// TIA Portal project "planta1_def_V15_V15.1" (V15.1)

(* hardware
DEVICE "S71500/ET200MP station_1"  S7-1500 station
   slot 0: "Perfil soporte_0"  Rack  6ES7 590-1***0-0AA0
   slot 1: "PLC_1"  CPU 1516-3 PN/DP  6ES7 516-3AN00-0AB0  V1.7
   slot 2: "DI 32x24VDC HF_1"  DI 32x24VDC HF  6ES7 521-1BL00-0AB0  V2.0
   slot 3: "DQ 32x24VDC/0.5A ST_1"  DQ 32x24VDC/0.5A ST  6ES7 522-1BL00-0AB0  V2.0
   slot 4: "AI 8xU/I/RTD/TC ST_1"  AI 8xU/I/RTD/TC ST  6ES7 531-7KF00-0AB0  V2.0
   slot 5: "AQ 4xU/I ST_1"  AQ 4xU/I ST  6ES7 532-5HD00-0AB0  V2.0
DEVICE "HMI_1"  TP1500 Comfort
   slot 0: "HMI"  HMI  6AV2 124-0QC02-0AX0  13.0.1.0
   slot 1: "HMI_RT_1"  TP1500 Comfort  6AV2 124-0QC02-0AX0  13.0.1.0
   slot 5: "HMI_1.IE_CP_1"  Interfaz PROFINET
      slot 1: "Interfaz PROFINET_1"  Interfaz PROFINET
         slot 1: "Port_1"  Port
         slot 2: "Port_2"  Port
   slot 6: "HMI_1.IE_CP_2"  Interfaz PROFINET
      slot 1: "Interfaz PROFINET_GBit"  Interfaz PROFINET
         slot 1: "Port_1"  Port
   slot 7: "HMI_1.MPI/DP_CP_1"  Interfaz MPI/DP
*)

// ===== PLC "PLC_1"  CPU 1516-3 PN/DP =====

VAR_GLOBAL   // PLC tag table "Tabla de variables estándar"
   "Switch de Nivel Bajo Tanque 1 (NO)" AT %I1.2 : Bool;   // OK
   "Switch de Nivel Alto Tanque 1 (NC)" AT %I1.3 : Bool;   // OK
   "Referencia Velocidad (VV)" AT %IW104 : Int;   // OK
   "Temperatura Liquido" AT %IW106 : Int;   // OK
   "Presión Liquido" AT %IW108 : Int;   // OK
   "Flujo Actual" AT %IW110 : Int;   // OK
   "Nivel tanque" AT %IW112 : Int;
   "Peso" AT %IW114 : Int;
   "FALLA (VF_DO2)" AT %I2.1 : Bool;   // Sin probar
   "Confirmación Celda BW31" AT %I2.6 : Bool;   // OK (Piloto por revisar)
   "ON/OFF1 (VF_DI1)" AT %Q2.0 : Bool;   // OK
   "Inversión (VF_DI2)" AT %Q2.1 : Bool;
   "Confirmación de Fallo (VF_DI3)" AT %Q2.2 : Bool;
   "Activar Unidad Calefactora" AT %Q1.6 : Bool;
   "RST Total1 (TF01)" AT %Q2.4 : Bool;   // OK
   "Siwarex DI0" AT %Q2.6 : Bool;
   "Siwarex DI1" AT %Q2.7 : Bool;
   "Abrir Valvula Llenado Tanque 1" AT %Q1.0 : Bool;   // OK
   "Abrir Valvula Vaciado Tanque 1" AT %Q1.1 : Bool;   // OK
   "Abrir Valvula Llenado Tanque 2" AT %Q1.2 : Bool;   // OK
   "Abrir Valvula Vaciado Tanque 2" AT %Q1.3 : Bool;   // OK
   "Abrir Valvula Llenado Tanque 3" AT %Q1.4 : Bool;   // OK
   "Abrir Valvula Vaciado Tanque 3" AT %Q1.5 : Bool;
   "Activar Unidad Enfriadora" AT %Q1.7 : Bool;   // OK
   "Panel de Mandos - Display 1" AT %QW100 : Int;
   "Panel de Mandos - Display 2" AT %QW102 : Int;
   "Consigna Velocidad Variador" AT %QW104 : Int;   // OK
   "Consigna apertura Valvula Proporcional" AT %QW106 : Int;   // OK
   "JOG Adelante (VF_DI4)" AT %Q2.3 : Bool;
   "System_Byte" AT %MB1 : Byte;
   "FirstScan" AT %M1.0 : Bool;
   "DiagStatusUpdate" AT %M1.1 : Bool;
   "AlwaysTRUE" AT %M1.2 : Bool;
   "AlwaysFALSE" AT %M1.3 : Bool;
   "Clock_Byte" AT %MB0 : Byte;
   "Clock_10Hz" AT %M0.0 : Bool;
   "Clock_5Hz" AT %M0.1 : Bool;
   "Clock_2.5Hz" AT %M0.2 : Bool;
   "Clock_2Hz" AT %M0.3 : Bool;
   "Clock_1.25Hz" AT %M0.4 : Bool;
   "Clock_1Hz" AT %M0.5 : Bool;
   "Clock_0.625Hz" AT %M0.6 : Bool;
   "Clock_0.5Hz" AT %M0.7 : Bool;
   "bomba" AT %MW6 : Int;
   "valvula" AT %MW8 : Int;
   "v1llen" AT %M2.3 : Bool;
   "v1vac" AT %M2.4 : Bool;
   "v2llen" AT %M2.5 : Bool;
   "v2vac" AT %M2.6 : Bool;
   "onproc" AT %M2.7 : Bool;
   "v3 vac" AT %M5.0 : Bool;
   "d7" AT %M3.0 : Bool;
   "presion" AT %MD10 : Real;
   "flujo" AT %MD14 : Real;
   "dfdf" AT %MD18 : Real;
   "encenderr" AT %M3.1 : Bool;
   "velmotor" AT %MW26 : Word;
   "Tag_19" AT %M3.2 : Bool;
   "onfuzz" AT %M5.1 : Bool;
   "onsint" AT %M5.3 : Bool;
   "onsmith" AT %M5.4 : Bool;
   "refsm" AT %MD20 : Real;
   "reffuzz" AT %MD22 : Real;
   "refsint" AT %MD24 : Real;
   "onsmtant" AT %M5.5 : Bool;
   "onlgr" AT %M5.6 : Bool;
   "reflgr" AT %MD26 : Real;
   "refsmtant" AT %MD28 : Real;
   "calefactora" AT %M6.0 : Bool;
   "Tag_21" AT %M6.1 : Bool;
   "enfriadora" AT %M7.0 : Bool;
   "temperatura" AT %MD16 : Real;
   "on_temp" AT %M5.7 : Bool;
   "REFTEMP" AT %MD30 : Real;
   "v3 llen" AT %M8.0 : Bool;
   "Tag_24" AT %MD50 : Real;
   "kp_sint" AT %MD34 : Real;
   "ki_sint" AT %MD38 : Real;
   "kd_sint" AT %MD42 : Real;
   "kp_lgr" AT %MD46 : Real;
   "ki_lgr" AT %MD54 : Real;
   "kd_lgr" AT %MD58 : Real;
   "kp_smith" AT %MD62 : Real;
   "ki_smith" AT %MD66 : Real;
   "kd_smith" AT %MD70 : Real;
   "kp_smitant" AT %MD74 : Real;
   "ki_smitant" AT %MD78 : Real;
   "kd_smitant" AT %MD82 : Real;
   "CERO_FUZ" AT %MD86 : Real;
   "POS_FUZZ" AT %MD90 : Real;
   "NEG_FUZZ" AT %MD94 : Real;
   "EN_1" AT %MD98 : Real;
   "EN_2" AT %MD102 : Real;
   "EN_3" AT %MD106 : Real;
   "EN_4" AT %MD110 : Real;
   "DEN_1" AT %MD114 : Real;
   "DEN_2" AT %MD118 : Real;
   "DEN_3" AT %MD122 : Real;
   "DEN_4" AT %MD126 : Real;
   "EZ_1" AT %MD130 : Real;
   "EZ_2" AT %MD134 : Real;
   "EZ_3" AT %MD138 : Real;
   "EZ_4" AT %MD142 : Real;
   "DEZ_1" AT %MD146 : Real;
   "DEZ_2" AT %MD150 : Real;
   "DEZ_3" AT %MD154 : Real;
   "DEZ_4" AT %MD158 : Real;
   "EP_1" AT %MD162 : Real;
   "EP_2" AT %MD166 : Real;
   "EP_3" AT %MD170 : Real;
   "EP_4" AT %MD174 : Real;
   "DEP_1" AT %MD178 : Real;
   "DEP_2" AT %MD182 : Real;
   "DEP_3" AT %MD186 : Real;
   "VARIADORFUZZ" AT %MD190 : Real;
   "DEP_4" AT %MD194 : Real;
   "ref_sint_presion" AT %MD198 : Real;
   "kp_sint_pres" AT %MD202 : Real;
   "ki_sint_presion" AT %MD206 : Real;
   "kd_sint_presion" AT %MD210 : Real;
   "on_sint_presion" AT %M2.0 : Bool;
   "on_lgr_flujo" AT %M2.1 : Bool;
   "ref_lgr_flujo" AT %MD214 : Real;
   "kp_lgr_flujo" AT %MD218 : Real;
   "ki_lgr_flujo" AT %MD222 : Real;
   "kd_lgr_flujo" AT %MD226 : Real;
   "onfuzz_presion" AT %M2.2 : Bool;
   "CERO_FUZ_presion" AT %MD230 : Real;
   "POS_FUZZ_presion" AT %MD234 : Real;
   "NEG_FUZZ_presion" AT %MD238 : Real;
   "EN_1_presion" AT %MD242 : Real;
   "EN_2_presion" AT %MD246 : Real;
   "EN_3_presion" AT %MD250 : Real;
   "EN_4_presion" AT %MD254 : Real;
   "DEN_1_presion" AT %MD258 : Real;
   "DEN_2_presion" AT %MD262 : Real;
   "DEN_3_presion" AT %MD266 : Real;
   "DEN_4_presion" AT %MD270 : Real;
   "EZ_1_presion" AT %MD274 : Real;
   "EZ_2_presion" AT %MD278 : Real;
   "EZ_3_presion" AT %MD282 : Real;
   "EZ_4_presion" AT %MD286 : Real;
   "DEZ_1_presion" AT %MD290 : Real;
   "DEZ_2_presion" AT %MD294 : Real;
   "DEZ_3_presion" AT %MD298 : Real;
   "DEZ_4_presion" AT %MD302 : Real;
   "EP_1_presion" AT %MD306 : Real;
   "EP_2_presion" AT %MD310 : Real;
   "EP_3_presion" AT %MD314 : Real;
   "EP_4_presion" AT %MD318 : Real;
   "DEP_1_presion" AT %MD322 : Real;
   "DEP_2_presion" AT %MD326 : Real;
   "DEP_3_presion" AT %MD330 : Real;
   "VARIADORFUZZ_presion" AT %MD334 : Real;
   "DEP_4_presion" AT %MD338 : Real;
   "reffuzz_presion" AT %MD342 : Real;
   "nivel_tanque" AT %MD346 : Real;
   "on_lgr_nivel" AT %M3.3 : Bool;
   "ref_lgr_nivel" AT %MD350 : Real;
   "kp_lgr_nivel" AT %MD354 : Real;
   "ki_lgr_nivel" AT %MD358 : Real;
   "kd_lgr_nivel" AT %MD362 : Real;
   "ALARMA1" AT %M200.0 : Bool;
   "ALARMA2" AT %M200.1 : Bool;
   "ALARMA3" AT %M200.3 : Bool;
   "on_nivel" AT %M3.4 : Bool;
   "ref_onoff_nivel" AT %MD366 : Real;
   "on_peso" AT %M3.5 : Bool;
   "peso tanque" AT %MD370 : Real;
   "ref_onoff_peso" AT %MD374 : Real;
   "Tag_1" AT %I2.3 : Bool;
   "Tag_2" AT %Q2.5 : Bool;
   "enclavar" AT %M3.6 : Bool;
   "Tag_3" AT %MW120 : Word;
   "Tag_4" AT %MD378 : Real;
   "Tag_5" AT %M100.4 : Bool;
   "Tag_6" AT %M100.5 : Bool;
   "Tag_7" AT %M100.6 : Bool;
   "M_Caracterizaicon" AT %M3.7 : Bool;
   "flujo_cal" AT %MD382 : Real;
   "presion_cal" AT %MD386 : Real;
   "temperatura_cal" AT %MD390 : Real;
   "nivel_cal" AT %MD394 : Real;
   "llenadot2" AT %M4.0 : Bool;
   "consigna_variador" AT %MW398 : Int;
   "iniciar_presion" AT %M4.1 : Bool;
   "llenadot1" AT %M4.2 : Bool;
   "ini_flujo" AT %M4.3 : Bool;
   "ini_temp" AT %M4.4 : Bool;
   "INICIAR_PID" AT %M4.5 : Bool;
   "sensor" AT %IW4 : Int;
   "sensor(1)" AT %IW6 : Int;
   "sensor(2)" AT %MW400 : Int;
   "act_calefactora" AT %M4.6 : Bool;
   "referen1" AT %MD402 : Real;
   "INICIAR_PIDP" AT %M4.7 : Bool;
   "Tag_8" AT %M33.0 : Bool;
   "Tag_9" AT %M18.1 : Bool;
   "Tag_10" AT %M18.2 : Bool;
   "Tag_11" AT %MD5 : Real;
   "Tag_12" AT %M71.0 : Bool;
   "Tag_13" AT %M12.0 : Bool;
   "Tag_14" AT %T1 : Timer;
   "Start" AT %M406.0 : Bool;
   "Tag_15" AT %M14.0 : Bool;
   "Tag_16" AT %M1.5 : Bool;
   "Tag_17" AT %QW20 : Word;
   "Tag_18" AT %MW20 : Word;
   "Tag_20" AT %T2 : Timer;
   "Tag_22" AT %MD100 : DWord;
   "Tag_23" AT %Q8.0 : Bool;
   "Tag_25" AT %MD101 : DWord;
   "Tag_26" AT %I2.0 : Bool;
   "Tag_27" AT %MD200 : Time;
   "Tag_28" AT %MD201 : Time;
   "Tag_29" AT %MD300 : Time;
   "Tag_30" AT %MD301 : Time;
   "activacion" AT %M406.1 : Bool;
   "u1" AT %MD408 : Real;
   "u2" AT %MD412 : Real;
   "e1" AT %MD416 : Real;
   "e2" AT %MD420 : Real;
   "rrr" AT %MD424 : Real;
   "activacion_smith_flujo" AT %M406.2 : Bool;
   "u3" AT %MD428 : Real;
   "u4" AT %MD432 : Real;
   "e3" AT %MD436 : Real;
   "e4" AT %MD440 : Real;
   "u1_1" AT %MD444 : Real;
   "u2_1" AT %MD448 : Real;
   "e1_1" AT %MD452 : Real;
   "e2_1" AT %MD456 : Real;
   "activacion_presion_si_es" AT %M406.3 : Bool;
   "referencia_fujo" AT %MD460 : Real;
   "activacion_filtro" AT %M406.4 : Bool;
   "presion_filtrada" AT %MD464 : Real;
   "e1f" AT %MD468 : Real;
   "e2f" AT %MD472 : Real;
   "u1f" AT %MD476 : Real;
   "u2f" AT %MD480 : Real;
   "activacion_flujo_definitivo" AT %M406.5 : Bool;
   "ref_presion" AT %MD484 : Real;
   "u11" AT %MD488 : Real;
   "u22" AT %MD492 : Real;
   "u33" AT %MD496 : Real;
   "u44" AT %MD500 : Real;
   "e11" AT %MD504 : Real;
   "e22" AT %MD508 : Real;
   "e33" AT %MD512 : Real;
   "e44" AT %MD516 : Real;
END_VAR

DATA_BLOCK "lgr_DB_1"   // DB1
{ S7_Optimized_Access := 'TRUE' }
VERSION : 0.1
// stored: InstanceOfName lgr
"lgr"
BEGIN
END_DATA_BLOCK

DATA_BLOCK "sintonizacion_DB_1"   // DB2
{ S7_Optimized_Access := 'TRUE' }
VERSION : 0.1
// stored: InstanceOfName sintonizacion
"sintonizacion"
BEGIN
END_DATA_BLOCK

DATA_BLOCK "smith_DB_2"   // DB3
{ S7_Optimized_Access := 'TRUE' }
VERSION : 0.1
// stored: InstanceOfName smith
"smith"
BEGIN
END_DATA_BLOCK

DATA_BLOCK "smithanticipativo_DB_1"   // DB4
{ S7_Optimized_Access := 'TRUE' }
VERSION : 0.1
// stored: InstanceOfName smithanticipativo
"smithanticipativo"
BEGIN
END_DATA_BLOCK

DATA_BLOCK "principal_DB"   // DB5
{ S7_Optimized_Access := 'TRUE' }
VERSION : 0.1
// stored: InstanceOfName principal
"principal"
BEGIN
END_DATA_BLOCK

DATA_BLOCK "lgr_DB_2"   // DB6
{ S7_Optimized_Access := 'TRUE' }
VERSION : 0.1
// stored: InstanceOfName lgr
"lgr"
BEGIN
END_DATA_BLOCK

DATA_BLOCK "ALARMA"   // DB7
{ S7_Optimized_Access := 'TRUE' }
VERSION : 0.1
   VAR
      ALARMA1 : Int;
      ALARMA2 : Int;
      ALARMA3 : Int;
      ALARMA4 : Int;
      ALARMA5 : Int;
      ALARMA6 : Int;
      ALARMA7 : Int;
      ALARMA8 : Int;
      ALARMA9 : Int;
      ALARMA10 : Int;
      ALARMA11 : Int;
      ALARMA12 : Int;
      ALARMA13 : Int;
      ALARMA14 : Int;
      ALARMA15 : Int;
      ALARMA16 : Int;
      ALARMA17 : Int;
      ALARMA18 : Int;
      ALARMA19 : Int;
      ALARMA20 : Int;
      ALARMA21 : Int;
      ALARMA22 : Int;
   END_VAR
BEGIN
END_DATA_BLOCK

DATA_BLOCK "DATOS_ENTRADAS_ANALOGAS"   // DB8
{ S7_Optimized_Access := 'TRUE' }
VERSION : 0.1
   VAR RETAIN
      "TRANSMISOR DE CAUDAL" : Struct   // Corriente 4 a 20 mA, 0 a 2000 l/h
         "LIMITE SUPERIOR" : Real := 2000.0;
         "LIMITE INFERIOR" : Real;
         AJUSTE : Real;
         "PUNTO INFERIOR" : Real;
         SOBRELIMITE : Bool;
         "ROTURA HILO" : Bool;
         "SEÑAL INGENIERIA" : Real;
      END_STRUCT;
      "TRANSMISOR DE PRESION" : Struct   // Corriente 4 a 20 mA, 0 a 36,25 psi
         "LIMITE SUPERIOR" : Real := 36.2594;   // 2,5 Bar = 36,2594 psi
         "LIMITE INFERIOR" : Real;
         AJUSTE : Real;
         "PUNTO INFERIOR" : Real;
         SOBRELIMITE : Bool;
         "ROTURA HILO" : Bool;
         "SEÑAL INGENIERIA" : Real;
      END_STRUCT;
      "TRANSMISOR DE TEMPERATURA" : Struct
         "LIMITE SUPERIOR" : Real := 100.0;
         "LIMITE INFERIOR" : Real;
         AJUSTE : Real;
         "PUNTO INFERIOR" : Real;
         SOBRELIMITE : Bool;
         "ROTURA HILO" : Bool;
         "SEÑAL INGENIERIA" : Real;
      END_STRUCT;
      "TRANSMISOR DE NIVEL" : Struct
         "LIMITE SUPERIOR" : Real := 100.0;
         "LIMITE INFERIOR" : Real;
         AJUSTE : Real;
         "PUNTO INFERIOR" : Real;
         SOBRELIMITE : Bool;
         "ROTURA HILO" : Bool;
         "SEÑAL INGENIERIA" : Real;
      END_STRUCT;
      "POTENCIOMETRO 1" : Struct   // Corriente 0 a 20 mA
         "LIMITE SUPERIOR" : Real := 20.0;
         "LIMITE INFERIOR" : Real;
         AJUSTE : Real;
         "PUNTO INFERIOR" : Real;
         SOBRELIMITE : Bool;
         "ROTURA HILO" : Bool;
         "SEÑAL INGENIERIA" : Real;
      END_STRUCT;
      "POTENCIOMETRO 2" : Struct   // Voltaje 0 a 10 V
         "LIMITE SUPERIOR" : Real := 10.0;
         "LIMITE INFERIOR" : Real;
         AJUSTE : Real;
         "PUNTO INFERIOR" : Real;
         SOBRELIMITE : Bool;
         "ROTURA HILO" : Bool;
         "SEÑAL INGENIERIA" : Real;
      END_STRUCT;
      VELOCIDAD_VARIADOR : Struct   // Corriente 4 a 20 mA, 0 a 100%
         "LIMITE SUPERIOR" : Real := 100.0;
         "LIMITE INFERIOR" : Real;
         AJUSTE : Real;
         "PUNTO INFERIOR" : Real;
         SOBRELIMITE : Bool;
         "ROTURA HILO" : Bool;
         "SEÑAL INGENIERIA" : Real;
      END_STRUCT;
   END_VAR
   VAR
      PESO : Struct   // Corriente 0 a 20 mA, 0 a 1,4 kg
         "LIMITE SUPERIOR" : Real := 1400.0;
         "LIMITE INFERIOR" : Real;
         AJUSTE : Real;
         "PUNTO INFERIOR" : Real;
         SOBRELIMITE : Bool;
         "ROTURA HILO" : Bool;
         "SEÑAL INGENIERIA" : Real;
      END_STRUCT;
   END_VAR
BEGIN
END_DATA_BLOCK

DATA_BLOCK "OnOff_nivel_DB"   // DB9
{ S7_Optimized_Access := 'TRUE' }
VERSION : 0.1
// stored: InstanceOfName OnOff_nivel
"OnOff_nivel"
BEGIN
END_DATA_BLOCK

DATA_BLOCK "DATOS_SALIDAS_ANALOGAS"   // DB10
{ S7_Optimized_Access := 'TRUE' }
VERSION : 0.1
   VAR RETAIN
      DISPLAY_1 : Struct
         "LIMITE INFERIOR" : Real := 4.0;
         "LIMITE SUPERIOR" : Real := 20.0;
         SEÑAL_INGENIERIA : Real;
         "REBASE POR EXCESO" : Bool;
      END_STRUCT;
      DISPLAY_2 : Struct
         "LIMITE INFERIOR" : Real;
         "LIMITE SUPERIOR" : Real := 10.0;
         SEÑAL_INGENIERIA : Real;
         "REBASE POR EXCESO" : Bool;
      END_STRUCT;
      "VALVULA PROPORCIONAL" : Struct
         "LIMITE INFERIOR" : Real;
         "LIMITE SUPERIOR" : Real := 100.0;
         SEÑAL_INGENIERIA : Real;
         "REBASE POR EXCESO" : Bool;
      END_STRUCT;
      VARIADOR : Struct
         "LIMITE INFERIOR" : Real;
         "LIMITE SUPERIOR" : Real := 100.0;
         SEÑAL_INGENIERIA : Real;
         "REBASE POR EXCESO" : Bool;
      END_STRUCT;
   END_VAR
BEGIN
END_DATA_BLOCK

DATA_BLOCK "pid NIVEL_DB"   // DB11
{ S7_Optimized_Access := 'TRUE' }
VERSION : 0.1
// stored: InstanceOfName pid NIVEL
"pid NIVEL"
BEGIN
END_DATA_BLOCK

DATA_BLOCK "OnOff_peso_DB"   // DB12
{ S7_Optimized_Access := 'TRUE' }
VERSION : 0.1
// stored: InstanceOfName OnOff_peso
"OnOff_peso"
BEGIN
END_DATA_BLOCK

DATA_BLOCK "VELOCIDAD_VARIADOR_FB_DB"   // DB13
{ S7_Optimized_Access := 'TRUE' }
VERSION : 0.1
// stored: InstanceOfName ENTRADAS_ANALOGAS_FB
"ENTRADAS_ANALOGAS_FB"
BEGIN
END_DATA_BLOCK

DATA_BLOCK "TEMPERATURA_FB_DB"   // DB14
{ S7_Optimized_Access := 'TRUE' }
VERSION : 0.1
// stored: InstanceOfName ENTRADAS_ANALOGAS_FB
"ENTRADAS_ANALOGAS_FB"
BEGIN
END_DATA_BLOCK

DATA_BLOCK "PRESION_LIQUIDO_FB_DB"   // DB15
{ S7_Optimized_Access := 'TRUE' }
VERSION : 0.1
// stored: InstanceOfName ENTRADAS_ANALOGAS_FB
"ENTRADAS_ANALOGAS_FB"
BEGIN
END_DATA_BLOCK

DATA_BLOCK "FLUJO_FB_DB"   // DB16
{ S7_Optimized_Access := 'TRUE' }
VERSION : 0.1
// stored: InstanceOfName ENTRADAS_ANALOGAS_FB
"ENTRADAS_ANALOGAS_FB"
BEGIN
END_DATA_BLOCK

DATA_BLOCK "NIVEL_FB_DB"   // DB17
{ S7_Optimized_Access := 'TRUE' }
VERSION : 0.1
// stored: InstanceOfName ENTRADAS_ANALOGAS_FB
"ENTRADAS_ANALOGAS_FB"
BEGIN
END_DATA_BLOCK

DATA_BLOCK "Caracterizacion_DB_1"   // DB18
{ S7_Optimized_Access := 'TRUE' }
VERSION : 0.1
// stored: InstanceOfName Caracterizacion
"Caracterizacion"
BEGIN
END_DATA_BLOCK

DATA_BLOCK "lgr_DB_3"   // DB19
{ S7_Optimized_Access := 'TRUE' }
VERSION : 0.1
// stored: InstanceOfName lgr
"lgr"
BEGIN
END_DATA_BLOCK

DATA_BLOCK "VELOCIDAD_VARIADOR_QW_FB_DB"   // DB20
{ S7_Optimized_Access := 'TRUE' }
VERSION : 0.1
// stored: InstanceOfName SALIDAS_ANALOGAS_FB
"SALIDAS_ANALOGAS_FB"
BEGIN
END_DATA_BLOCK

DATA_BLOCK "VALVULA_PROPORCIONAL_FB_DB"   // DB21
{ S7_Optimized_Access := 'TRUE' }
VERSION : 0.1
// stored: InstanceOfName SALIDAS_ANALOGAS_FB
"SALIDAS_ANALOGAS_FB"
BEGIN
END_DATA_BLOCK

DATA_BLOCK "Calibracion Flujo_DB_1"   // DB22
{ S7_Optimized_Access := 'TRUE' }
VERSION : 0.1
// stored: InstanceOfName Calibracion Flujo
"Calibracion Flujo"
BEGIN
END_DATA_BLOCK

DATA_BLOCK "lgr_DB_4"   // DB23
{ S7_Optimized_Access := 'TRUE' }
VERSION : 0.1
// stored: InstanceOfName lgr
"lgr"
BEGIN
END_DATA_BLOCK

DATA_BLOCK "Bloque_2_DB"   // DB24
{ S7_Optimized_Access := 'TRUE' }
VERSION : 0.1
// stored: InstanceOfName Bloque_2
"Bloque_2"
BEGIN
END_DATA_BLOCK

DATA_BLOCK "Bloque_2_DB_1"   // DB25
{ S7_Optimized_Access := 'TRUE' }
VERSION : 0.1
// stored: InstanceOfName Bloque_2
"Bloque_2"
BEGIN
END_DATA_BLOCK

DATA_BLOCK "Bloque_2_DB_2"   // DB26
{ S7_Optimized_Access := 'TRUE' }
VERSION : 0.1
// stored: InstanceOfName Bloque_2
"Bloque_2"
BEGIN
END_DATA_BLOCK

DATA_BLOCK "Bloque_2_DB_4"   // DB27
{ S7_Optimized_Access := 'TRUE' }
VERSION : 0.1
// stored: InstanceOfName Bloque_2
"Bloque_2"
BEGIN
END_DATA_BLOCK

DATA_BLOCK "Bloque_2_DB_3"   // DB28
{ S7_Optimized_Access := 'TRUE' }
VERSION : 0.1
// stored: InstanceOfName Bloque_2
"Bloque_2"
BEGIN
END_DATA_BLOCK

DATA_BLOCK "FlujoSergioCortes_DB"   // DB29
{ S7_Optimized_Access := 'TRUE' }
VERSION : 0.1
// stored: InstanceOfName PID_FLUJO
"PID_FLUJO"
BEGIN
END_DATA_BLOCK

DATA_BLOCK "FlujoSergioCortes_DB_1"   // DB30
{ S7_Optimized_Access := 'TRUE' }
VERSION : 0.1
// stored: InstanceOfName PID_FLUJO
"PID_FLUJO"
BEGIN
END_DATA_BLOCK

DATA_BLOCK "Bloque_2_DB_5"   // DB31
{ S7_Optimized_Access := 'TRUE' }
VERSION : 0.1
// stored: InstanceOfName Bloque_2
"Bloque_2"
BEGIN
END_DATA_BLOCK

DATA_BLOCK "Bloque_2_DB_6"   // DB33
{ S7_Optimized_Access := 'TRUE' }
VERSION : 0.1
// stored: InstanceOfName Bloque_2
"Bloque_2"
BEGIN
END_DATA_BLOCK

DATA_BLOCK "PESO_FB_DB"   // DB34
{ S7_Optimized_Access := 'TRUE' }
VERSION : 0.1
// stored: InstanceOfName ENTRADAS_ANALOGAS_FB
"ENTRADAS_ANALOGAS_FB"
BEGIN
END_DATA_BLOCK

DATA_BLOCK "FlujoSergioCortes_DB_2"   // DB35
{ S7_Optimized_Access := 'TRUE' }
VERSION : 0.1
// stored: InstanceOfName PID_FLUJO
"PID_FLUJO"
BEGIN
END_DATA_BLOCK

DATA_BLOCK "Bloque_2_DB_7"   // DB36
{ S7_Optimized_Access := 'TRUE' }
VERSION : 0.1
// stored: InstanceOfName Bloque_2
"Bloque_2"
BEGIN
END_DATA_BLOCK

DATA_BLOCK "fuzzyficacion_DB"   // DB37
{ S7_Optimized_Access := 'TRUE' }
VERSION : 0.1
// stored: InstanceOfName fuzzyficacion
"fuzzyficacion"
BEGIN
END_DATA_BLOCK

DATA_BLOCK "FUZZY"   // DB38
{ S7_Optimized_Access := 'TRUE' }
VERSION : 0.1
// stored: InstanceOfName principal
"principal"
BEGIN
END_DATA_BLOCK

DATA_BLOCK "smith_DB"   // DB39
{ S7_Optimized_Access := 'TRUE' }
VERSION : 0.1
// stored: InstanceOfName smith
"smith"
BEGIN
END_DATA_BLOCK

DATA_BLOCK "smith_DB_1"   // DB40
{ S7_Optimized_Access := 'TRUE' }
VERSION : 0.1
// stored: InstanceOfName smith
"smith"
BEGIN
END_DATA_BLOCK

DATA_BLOCK "smithanticipativo_DB"   // DB41
{ S7_Optimized_Access := 'TRUE' }
VERSION : 0.1
// stored: InstanceOfName smithanticipativo
"smithanticipativo"
BEGIN
END_DATA_BLOCK

DATA_BLOCK "lgr_DB"   // DB42
{ S7_Optimized_Access := 'TRUE' }
VERSION : 0.1
// stored: InstanceOfName lgr
"lgr"
BEGIN
END_DATA_BLOCK

DATA_BLOCK "controltemperatura_DB"   // DB43
{ S7_Optimized_Access := 'TRUE' }
VERSION : 0.1
// stored: InstanceOfName controltemperatura
"controltemperatura"
BEGIN
END_DATA_BLOCK

DATA_BLOCK "FlujoSergioCortes_DB_3"   // DB44
{ S7_Optimized_Access := 'TRUE' }
VERSION : 0.1
// stored: InstanceOfName PID_FLUJO
"PID_FLUJO"
BEGIN
END_DATA_BLOCK

DATA_BLOCK "Calibracion Presion_DB_1"   // DB45
{ S7_Optimized_Access := 'TRUE' }
VERSION : 0.1
// stored: InstanceOfName Calibracion Presion
"Calibracion Presion"
BEGIN
END_DATA_BLOCK

DATA_BLOCK "Calibracion temperatura_DB_1"   // DB46
{ S7_Optimized_Access := 'TRUE' }
VERSION : 0.1
// stored: InstanceOfName Calibracion temperatura
"Calibracion temperatura"
BEGIN
END_DATA_BLOCK

DATA_BLOCK "Calibracion_Nivel_DB_1"   // DB47
{ S7_Optimized_Access := 'TRUE' }
VERSION : 0.1
// stored: InstanceOfName Calibracion_Nivel
"Calibracion_Nivel"
BEGIN
END_DATA_BLOCK

DATA_BLOCK "Caracterizacion_DB"   // DB48
{ S7_Optimized_Access := 'TRUE' }
VERSION : 0.1
// stored: InstanceOfName Caracterizacion
"Caracterizacion"
BEGIN
END_DATA_BLOCK

DATA_BLOCK "Calibracion_Nivel_DB"   // DB49
{ S7_Optimized_Access := 'TRUE' }
VERSION : 0.1
// stored: InstanceOfName Calibracion_Nivel
"Calibracion_Nivel"
BEGIN
END_DATA_BLOCK

DATA_BLOCK "Calibracion Presion_DB"   // DB50
{ S7_Optimized_Access := 'TRUE' }
VERSION : 0.1
// stored: InstanceOfName Calibracion Presion
"Calibracion Presion"
BEGIN
END_DATA_BLOCK

DATA_BLOCK "Calibracion temperatura_DB"   // DB51
{ S7_Optimized_Access := 'TRUE' }
VERSION : 0.1
// stored: InstanceOfName Calibracion temperatura
"Calibracion temperatura"
BEGIN
END_DATA_BLOCK

DATA_BLOCK "Calibracion Flujo_DB"   // DB52
{ S7_Optimized_Access := 'TRUE' }
VERSION : 0.1
// stored: InstanceOfName Calibracion Flujo
"Calibracion Flujo"
BEGIN
END_DATA_BLOCK

DATA_BLOCK "PID_FLUJO_DB"   // DB53
{ S7_Optimized_Access := 'TRUE' }
VERSION : 0.1
// stored: InstanceOfName PID_FLUJO
"PID_FLUJO"
BEGIN
END_DATA_BLOCK

DATA_BLOCK "PID_FLUJO_DB_1"   // DB54
{ S7_Optimized_Access := 'TRUE' }
VERSION : 0.1
// stored: InstanceOfName PID_FLUJO
"PID_FLUJO"
BEGIN
END_DATA_BLOCK

DATA_BLOCK "PID_FLUJO_DB_2"   // DB55
{ S7_Optimized_Access := 'TRUE' }
VERSION : 0.1
// stored: InstanceOfName PID_FLUJO
"PID_FLUJO"
BEGIN
END_DATA_BLOCK

DATA_BLOCK "PID_PRESION_DB"   // DB56
{ S7_Optimized_Access := 'TRUE' }
VERSION : 0.1
// stored: InstanceOfName PID_PRESION
"PID_PRESION"
BEGIN
END_DATA_BLOCK

DATA_BLOCK "smith completo_DB"   // DB57
{ S7_Optimized_Access := 'TRUE' }
VERSION : 0.1
// stored: InstanceOfName smith completo
"smith completo"
BEGIN
END_DATA_BLOCK

DATA_BLOCK "Smith_please_DB"   // DB58
{ S7_Optimized_Access := 'TRUE' }
VERSION : 0.1
// stored: InstanceOfName Smith_please
"Smith_please"
BEGIN
END_DATA_BLOCK

DATA_BLOCK "Smith_please_DB_1"   // DB59
{ S7_Optimized_Access := 'TRUE' }
VERSION : 0.1
// stored: InstanceOfName Smith_please
"Smith_please"
BEGIN
END_DATA_BLOCK

DATA_BLOCK "CAUDAL"   // DB61
{ S7_Optimized_Access := 'TRUE' }
VERSION : 0.1
   VAR
      NIVELT : Array[0..20] of Real;
      NIVELT2 : Array[0..20] of Real;
      FLUJO : Array[0..20] of Real;
   END_VAR
BEGIN
END_DATA_BLOCK

DATA_BLOCK "CALCULO_FLUJO_DB"   // DB65
{ S7_Optimized_Access := 'TRUE' }
VERSION : 0.1
// stored: InstanceOfName CALCULO_FLUJO
"CALCULO_FLUJO"
BEGIN
END_DATA_BLOCK

DATA_BLOCK "DELTA_NIVEL"   // DB66
{ S7_Optimized_Access := 'TRUE' }
VERSION : 0.1
   VAR
      N1 : Real;
      N2 : Real;
      FLUJO : Array[0..50] of Real;
      flujoplc : Array[0..50] of Real;
      DELTA : Real;
   END_VAR
BEGIN
END_DATA_BLOCK

DATA_BLOCK "PresionZd"   // DB69
{ S7_Optimized_Access := 'TRUE' }
VERSION : 0.1
   VAR
      e1 : Real := 0.0;
      e2 : Real := 0.0;
      e3 : Real := 0.0;
      e4 : Real := 0.0;
      e5 : Real := 0.0;
      u1 : Real := 0.0;
      u2 : Real := 0.0;
      u3 : Real := 0.0;
      u4 : Real := 0.0;
      u5 : Real := 0.0;
      ud1 : Real := 0.0;
      ud2 : Real := 0.0;
      ds1 : Real := 0.0;
      ds2 : Real := 0.0;
   END_VAR
BEGIN
END_DATA_BLOCK

DATA_BLOCK "PID_FLUJO_DB_3"   // DB70
{ S7_Optimized_Access := 'TRUE' }
VERSION : 0.1
// stored: InstanceOfName PID_FLUJO
"PID_FLUJO"
BEGIN
END_DATA_BLOCK

DATA_BLOCK "PID_JyH_DB"   // DB71
{ S7_Optimized_Access := 'TRUE' }
VERSION : 0.1
// stored: InstanceOfName PID_JyH
"PID_JyH"
BEGIN
END_DATA_BLOCK

DATA_BLOCK "Smith Flujo_DB"   // DB72
{ S7_Optimized_Access := 'TRUE' }
VERSION : 0.1
// stored: InstanceOfName Smith Flujo
"Smith Flujo"
BEGIN
END_DATA_BLOCK

DATA_BLOCK "Smith Flujo_1_DB"   // DB73
{ S7_Optimized_Access := 'TRUE' }
VERSION : 0.1
// stored: InstanceOfName Smith Presion
"Smith Presion"
BEGIN
END_DATA_BLOCK

DATA_BLOCK "Smith Flujo_DB_1"   // DB74
{ S7_Optimized_Access := 'TRUE' }
VERSION : 0.1
// stored: InstanceOfName Smith Flujo
"Smith Flujo"
BEGIN
END_DATA_BLOCK

DATA_BLOCK "smith_flujo_definitivo_DB"   // DB75
{ S7_Optimized_Access := 'TRUE' }
VERSION : 0.1
// stored: InstanceOfName smith_flujo_definitivo
"smith_flujo_definitivo"
BEGIN
END_DATA_BLOCK

DATA_BLOCK "filto_DB"   // DB76
{ S7_Optimized_Access := 'TRUE' }
VERSION : 0.1
// stored: InstanceOfName filto
"filto"
BEGIN
END_DATA_BLOCK

DATA_BLOCK "smith_presion_definitivo_DB"   // DB77
{ S7_Optimized_Access := 'TRUE' }
VERSION : 0.1
// stored: InstanceOfName smith_presion_definitivo
"smith_presion_definitivo"
BEGIN
END_DATA_BLOCK

// folder: System blocks/Program resources

DATA_BLOCK "IEC_Counter_ml_DB"   // DB32
{ S7_Optimized_Access := 'TRUE' }
AUTHOR : SIMATIC
FAMILY : IEC
NAME : DCNTR
VERSION : 1.2
// stored: InstanceOfName IEC_DCOUNTER
"IEC_DCOUNTER"
BEGIN
END_DATA_BLOCK

DATA_BLOCK "IEC_Timer_0_DB"   // DB60
{ S7_Optimized_Access := 'TRUE' }
AUTHOR : Simatic
FAMILY : IEC
NAME : IEC_TMR
VERSION : 1.0
// stored: InstanceOfName IEC_TIMER
"IEC_TIMER"
BEGIN
END_DATA_BLOCK

DATA_BLOCK "IEC_Timer_0_DB_1"   // DB62
{ S7_Optimized_Access := 'TRUE' }
AUTHOR : Simatic
FAMILY : IEC
NAME : IEC_TMR
VERSION : 1.0
// stored: InstanceOfName IEC_TIMER
"IEC_TIMER"
BEGIN
END_DATA_BLOCK

DATA_BLOCK "IEC_Timer_0_DB_2"   // DB63
{ S7_Optimized_Access := 'TRUE' }
AUTHOR : Simatic
FAMILY : IEC
NAME : IEC_TMR
VERSION : 1.0
// stored: InstanceOfName IEC_TIMER
"IEC_TIMER"
BEGIN
END_DATA_BLOCK

DATA_BLOCK "IEC_Timer_0_DB_3"   // DB64
{ S7_Optimized_Access := 'TRUE' }
AUTHOR : Simatic
FAMILY : IEC
NAME : IEC_TMR
VERSION : 1.0
// stored: InstanceOfName IEC_TIMER
"IEC_TIMER"
BEGIN
END_DATA_BLOCK

DATA_BLOCK "IEC_Timer_0_DB_4"   // DB67
{ S7_Optimized_Access := 'TRUE' }
AUTHOR : Simatic
FAMILY : IEC
NAME : IEC_TMR
VERSION : 1.0
// stored: InstanceOfName IEC_TIMER
"IEC_TIMER"
BEGIN
END_DATA_BLOCK

DATA_BLOCK "IEC_Timer_0_DB_5"   // DB68
{ S7_Optimized_Access := 'TRUE' }
AUTHOR : Simatic
FAMILY : IEC
NAME : IEC_TMR
VERSION : 1.0
// stored: InstanceOfName IEC_TIMER
"IEC_TIMER"
BEGIN
END_DATA_BLOCK

// folder: (top level)

FUNCTION_BLOCK "ENTRADAS_ANALOGAS_FB"   // FB1, LAD
{ S7_Optimized_Access := 'TRUE' }
VERSION : 0.1
   VAR_INPUT
      SEÑAL_PERIFERIA : Int;
      LIMITE_SUPERIOR : Real;
      LIMITE_INFERIOR : Real;
      AJUSTE : Real := 0.0;
      PUNTO_INFERIOR : Real;
   END_VAR
   VAR_OUTPUT
      SEÑAL_INGENIERIA : Real;
      SOBRE_LÍMITE : Bool;
      ROTURA_HILO : Bool;
   END_VAR
   VAR
      SEÑAL_REAL : Real;
      TEMP1 : Real;
      TEMP2 : Real;
      PENDIENTE : Real;
      MX : Real;
      "MX+B" : Real;
      SEÑAL_CORREGIDA : Real;
   END_VAR
BEGIN

REGION Network 1
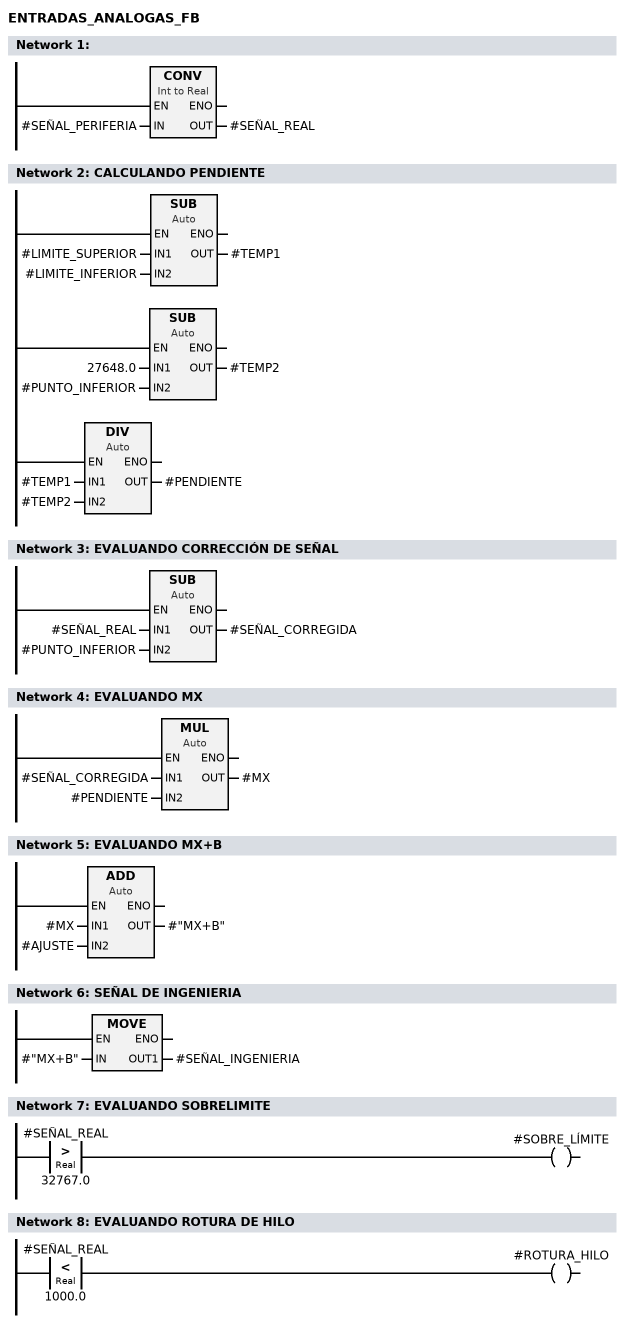
   RUNG wire#powerrail
      { S7_Templates := "[SrcType := Int, DestType := Real]" } Convert(in := #SEÑAL_PERIFERIA, out => #SEÑAL_REAL)
   END_RUNG
   // the same network as SCL:
   #SEÑAL_REAL := INT_TO_REAL(#SEÑAL_PERIFERIA);
END_REGION

REGION Network 2: CALCULANDO PENDIENTE
   RUNG wire#powerrail
      Sub(in1 := #LIMITE_SUPERIOR, in2 := #LIMITE_INFERIOR, out => #TEMP1)
   END_RUNG
   RUNG wire#powerrail
      Sub(in1 := 27648.0, in2 := #PUNTO_INFERIOR, out => #TEMP2)
   END_RUNG
   RUNG wire#powerrail
      Div(in1 := #TEMP1, in2 := #TEMP2, out => #PENDIENTE)
   END_RUNG
   // the same network as SCL:
   #TEMP1 := #LIMITE_SUPERIOR - #LIMITE_INFERIOR;
   #TEMP2 := 27648.0 - #PUNTO_INFERIOR;
   #PENDIENTE := #TEMP1 / #TEMP2;
END_REGION

REGION Network 3: EVALUANDO CORRECCIÓN DE SEÑAL
   RUNG wire#powerrail
      Sub(in1 := #SEÑAL_REAL, in2 := #PUNTO_INFERIOR, out => #SEÑAL_CORREGIDA)
   END_RUNG
   // the same network as SCL:
   #SEÑAL_CORREGIDA := #SEÑAL_REAL - #PUNTO_INFERIOR;
END_REGION

REGION Network 4: EVALUANDO MX
   RUNG wire#powerrail
      Mul(in1 := #SEÑAL_CORREGIDA, in2 := #PENDIENTE, out => #MX)
   END_RUNG
   // the same network as SCL:
   #MX := #SEÑAL_CORREGIDA * #PENDIENTE;
END_REGION

REGION Network 5: EVALUANDO MX+B
   RUNG wire#powerrail
      Add(in1 := #MX, in2 := #AJUSTE, out => #"MX+B")
   END_RUNG
   // the same network as SCL:
   #"MX+B" := #MX + #AJUSTE;
END_REGION

REGION Network 6: SEÑAL DE INGENIERIA
   RUNG wire#powerrail
      Move(in := #"MX+B", out1 => #SEÑAL_INGENIERIA)
   END_RUNG
   // the same network as SCL:
   #SEÑAL_INGENIERIA := #"MX+B";
END_REGION

REGION Network 7: EVALUANDO SOBRELIMITE
   RUNG wire#powerrail
      { S7_Templates := "SrcType := Real" } GT_Contact(in1 := #SEÑAL_REAL, in2 := 32767.0)
      Coil( #SOBRE_LÍMITE )
   END_RUNG
   // the same network as SCL:
   #SOBRE_LÍMITE := #SEÑAL_REAL > 32767.0;
END_REGION

REGION Network 8: EVALUANDO ROTURA DE HILO
   RUNG wire#powerrail
      { S7_Templates := "SrcType := Real" } LT_Contact(in1 := #SEÑAL_REAL, in2 := 1000.0)
      Coil( #ROTURA_HILO )
   END_RUNG
   // the same network as SCL:
   #ROTURA_HILO := #SEÑAL_REAL < 1000.0;
END_REGION
END_FUNCTION_BLOCK

FUNCTION_BLOCK "SALIDAS_ANALOGAS_FB"   // FB2, LAD
{ S7_Optimized_Access := 'TRUE' }
VERSION : 0.1
   VAR_INPUT
      "SEÑAL INGENIERIA" : Real;
      "LIMITE SUPERIOR" : Real;
      "LIMITE INFERIOR" : Real;
      "PUNTO INFERIOR" : Real;
   END_VAR
   VAR_OUTPUT
      "SEÑAL PERIFERIA" : Int;
      "REBASE POR EXCESO" : Bool;
   END_VAR
   VAR_TEMP
      TEMP_1 : Real;
      TEMP_2 : Real;
      TEMP_3 : Real;
      TEMP_4 : Real;
      TEMP_5 : Real;
      K1 : Real;
      K2 : Real;
      SEÑAL_REAL : Real;
   END_VAR
BEGIN

REGION Network 1
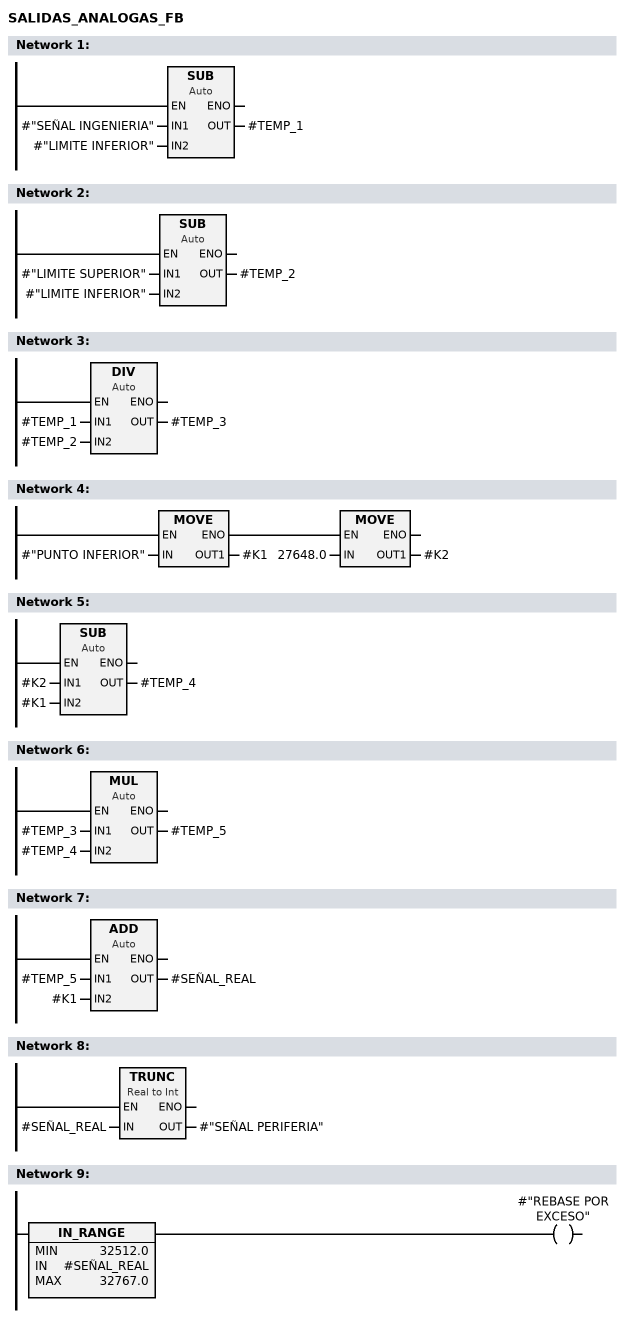
   RUNG wire#powerrail
      Sub(in1 := #"SEÑAL INGENIERIA", in2 := #"LIMITE INFERIOR", out => #TEMP_1)
   END_RUNG
   // the same network as SCL:
   #TEMP_1 := #"SEÑAL INGENIERIA" - #"LIMITE INFERIOR";
END_REGION

REGION Network 2
   RUNG wire#powerrail
      Sub(in1 := #"LIMITE SUPERIOR", in2 := #"LIMITE INFERIOR", out => #TEMP_2)
   END_RUNG
   // the same network as SCL:
   #TEMP_2 := #"LIMITE SUPERIOR" - #"LIMITE INFERIOR";
END_REGION

REGION Network 3
   RUNG wire#powerrail
      Div(in1 := #TEMP_1, in2 := #TEMP_2, out => #TEMP_3)
   END_RUNG
   // the same network as SCL:
   #TEMP_3 := #TEMP_1 / #TEMP_2;
END_REGION

REGION Network 4
   RUNG wire#powerrail
      Move(in := #"PUNTO INFERIOR", out1 => #K1)
      Move(in := 27648.0, out1 => #K2)
   END_RUNG
   // the same network as SCL:
   #K1 := #"PUNTO INFERIOR";
   #K2 := 27648.0;
END_REGION

REGION Network 5
   RUNG wire#powerrail
      Sub(in1 := #K2, in2 := #K1, out => #TEMP_4)
   END_RUNG
   // the same network as SCL:
   #TEMP_4 := #K2 - #K1;
END_REGION

REGION Network 6
   RUNG wire#powerrail
      Mul(in1 := #TEMP_3, in2 := #TEMP_4, out => #TEMP_5)
   END_RUNG
   // the same network as SCL:
   #TEMP_5 := #TEMP_3 * #TEMP_4;
END_REGION

REGION Network 7
   RUNG wire#powerrail
      Add(in1 := #TEMP_5, in2 := #K1, out => #SEÑAL_REAL)
   END_RUNG
   // the same network as SCL:
   #SEÑAL_REAL := #TEMP_5 + #K1;
END_REGION

REGION Network 8
   RUNG wire#powerrail
      { S7_Templates := "[SrcType := Real, DestType := Int]" } Trunc(in := #SEÑAL_REAL, out => #"SEÑAL PERIFERIA")
   END_RUNG
   // the same network as SCL:
   #"SEÑAL PERIFERIA" := TRUNC(#SEÑAL_REAL);
END_REGION

REGION Network 9
   RUNG wire#powerrail
      { S7_Templates := "SrcType := Real" } InRange(min := 32512.0, in := #SEÑAL_REAL, max := 32767.0)
      Coil( #"REBASE POR EXCESO" )
   END_RUNG
   // the same network as SCL:
   #"REBASE POR EXCESO" := (32512.0 <= #SEÑAL_REAL) AND (#SEÑAL_REAL <= 32767.0);
END_REGION
END_FUNCTION_BLOCK

FUNCTION_BLOCK "MAG5100W"   // FB3, LAD
{ S7_Optimized_Access := 'TRUE' }
VERSION : 0.1
   VAR_INPUT
      "Q(ml)" : Bool;
      "OK(Batch)" : Bool;
   END_VAR
   VAR_OUTPUT
      Zero : Bool;
   END_VAR
   VAR
      Reset : Bool;
      FP : Bool;
      Fin_Batch : Bool;
      R_Total_1 : Bool;
      "No(100ml)" : DInt := 10;
      Preset : DInt := 100;
   END_VAR
   VAR_TEMP   // added for the SCL form of the ladder/FBD networks
      _w1 : Bool;
   END_VAR
BEGIN

REGION Network 1
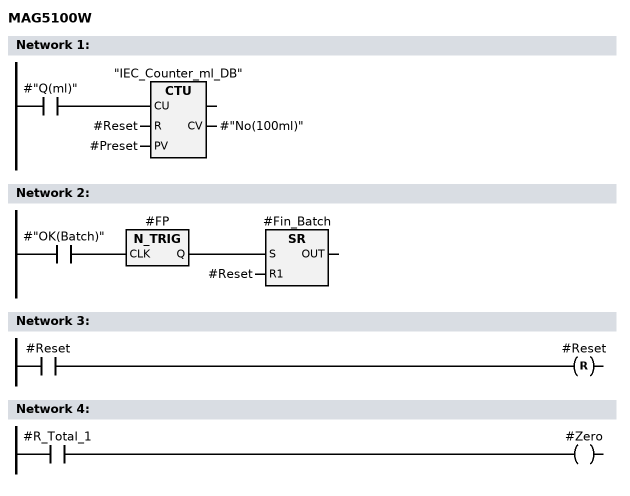
   "IEC_Counter_ml_DB".CTU(CU := #"Q(ml)", R := #Reset, PV := #Preset, CV => #"No(100ml)");
END_REGION

REGION Network 2
   RUNG wire#powerrail
      Contact( #"OK(Batch)" )
      N_Trig( #FP )
      S_SR(operand := #Fin_Batch, r1 := #Reset)
   END_RUNG
   // the same network as SCL:
   #_w1 := NOT #"OK(Batch)" AND #FP;   // falling edge
   #FP := #"OK(Batch)";
   IF #_w1 THEN
       #Fin_Batch := TRUE;   // SR flip-flop
   END_IF;
   IF #Reset THEN #Fin_Batch := FALSE; END_IF;
END_REGION

REGION Network 3
   RUNG wire#powerrail
      Contact( #Reset )
      R_Coil( #Reset )
   END_RUNG
   // the same network as SCL:
   IF #Reset THEN #Reset := FALSE; END_IF;
END_REGION

REGION Network 4
   RUNG wire#powerrail
      Contact( #R_Total_1 )
      Coil( #Zero )
   END_RUNG
   // the same network as SCL:
   #Zero := #R_Total_1;
END_REGION
END_FUNCTION_BLOCK

FUNCTION_BLOCK "sintonizacion"   // FB4, SCL
{ S7_Optimized_Access := 'TRUE' }
VERSION : 0.1
   VAR_INPUT
      ref : Real;
      kp : Real := 30.0;
      ki : Real := 3.0;
      kd : Real := 0.5;
      sensor : Real;
   END_VAR
   VAR_OUTPUT
      señal_u : Real;
      error : Real;
      e0 : Real;
      de : Real;
      e1 : Real;
   END_VAR
BEGIN
   #error := #ref - #sensor;
   #e1 :=  #e1 +#error * 0.01;//periodo de muestreo t
   #de := (#error - #e0) / 0.01;
   //7.2722 49.6172;

   #señal_u := (#kp * #error + #ki * #e1 + #de * #kd);
   IF #señal_u > 27000.0 THEN
       #señal_u := 27000.0;
   END_IF;
   IF #señal_u < 9000.0 THEN
       #señal_u := 9000.0;
   END_IF;
END_FUNCTION_BLOCK

FUNCTION_BLOCK "fuzzyficacion"   // FB5, SCL
{ S7_Optimized_Access := 'TRUE' }
VERSION : 0.1
   VAR_INPUT
      crisp : Real;
      vector1 : Real;
      vector2 : Real;
      vector3 : Real;
      vector4 : Real;
   END_VAR
   VAR_OUTPUT
      S : Real;
   END_VAR
   VAR_TEMP
      "a" : Real;
      "B" : Real;
   END_VAR
BEGIN
   IF (#vector1 < #crisp & #crisp < #vector2) THEN
       #B := -1 * (((1 - 0) / (#vector2 - #vector1)) * #vector1);
       #a := (((1 - 0) / (#vector2 - #vector1)) * #crisp) + #B;
   END_IF;
   IF (#vector2 < #crisp & #crisp < #vector3) THEN
       #a := 1;
   END_IF;
   IF (#vector3 < #crisp & #crisp < #vector4) THEN
       #B := (((1 - 0) / (#vector2 - #vector1)) * #vector4);
       #a := (((0 - 1) / (#vector4 - #vector3)) * #crisp) + #B;
   ELSE
       #a := 0;
   END_IF;
   #S := #a;
END_FUNCTION_BLOCK

FUNCTION_BLOCK "principal"   // FB6, SCL
{ S7_Optimized_Access := 'TRUE' }
VERSION : 0.1
   VAR_INPUT
      sensor : Real;
      ki : Real := 15.0;
      Z : Real := 0.0;
      P : Real := 9730.0;
      N : Real := -9730.0;
      EN1 : Real := -688.0;
      EN2 : Real := -432.0;
      EN3 : Real := -294.8;
      EN4 : Real := -41.3;
      DEN1 : Real := -783.0;
      DEN2 : Real := -607.0;
      DEN3 : Real := -364.1;
      DEN4 : Real := -63.3;
      EZ1 : Real := -103.0;
      EZ2 : Real := -10.0;
      EZ3 : Real := 10.0;
      EZ4 : Real := 104.8;
      DEZ1 : Real := -93.6;
      DEZ2 : Real := -10.4;
      DEZ3 : Real := 10.45;
      DEZ4 : Real := 94.05;
      EP1 : Real := 43.4;
      EP2 : Real := 296.5;
      EP3 : Real := 432.0;
      EP4 : Real := 688.0;
      DEP1 : Real := 11.22;
      DEP2 : Real := 347.0;
      DEP3 : Real := 544.0;
      var : Real := 9000.0;
      DEP4 : Real := 812.0;
      ref : Real;
   END_VAR
   VAR_OUTPUT
      S : Real;
      "e" : Real;
      de : Real;
   END_VAR
   VAR_TEMP
      R1 : Real;
      R2 : Real;
      R3 : Real;
      R4 : Real;
      R5 : Real;
      R6 : Real;
      R7 : Real;
      R8 : Real;
      R9 : Real;
      e0 : Real;
      AA : Real;
      BB : Real;
      eant : Real;
      SS : Real;
      e1 : Real;
      pi : Real;
      CC : Real;
   END_VAR
BEGIN
   #e := #ref - #sensor;
   #de := (#e-#eant);
   #e1 := #e1 + #e;
   #pi := #e1 *#ki;
   #eant := #e;"fuzzyfica"(crisp := #e,
               vector1 := #EN1,
               vector2 := #EN2,
               vector3 := #EN3,
               vector4 := #EN4,
               A_1 => #AA);
   "fuzzyfica" (crisp := #de,
                                     vector1 := #DEN1,
                                     vector2 := #DEN2,
                                     vector3 := #DEN3,
                                     vector4 := #DEN4,
                                     A_1 => #BB);
   #R1:=MIN_REAL(IN1:=#AA,IN2:=#BB);
   "fuzzyfica"(crisp := #e,
                                    vector1 := #EN1,
                                    vector2 := #EN2,
                                    vector3 := #EN3,
                                    vector4 := #EN4,
                                    A_1 => #AA);
   "fuzzyfica"(crisp := #de,
                                    vector1 := #DEZ1,
                                    vector2 := #DEZ2,
                                    vector3 := #DEZ3,
                                    vector4 := #DEZ4,
                                    A_1 => #BB);
   #R2 := MIN_REAL(IN1 := #AA, IN2 := #BB);
   "fuzzyfica"(crisp := #e,
                                    vector1 := #EN1,
                                    vector2 := #EN2,
                                    vector3 := #EN3,
                                    vector4 := #EN4,
                                    A_1 => #AA);
   "fuzzyfica"(crisp := #de,
                                    vector1 := #DEP1,
                                    vector2 := #DEP2,
                                    vector3 := #DEP3,
                                    vector4 := #DEP4,
                                    A_1 => #BB);
   #R3 := MIN_REAL(IN1 := #AA, IN2 := #BB);
   "fuzzyfica"(crisp := #e,
                                    vector1 := #EZ1,
                                    vector2 := #EZ2,
                                    vector3 := #EZ3,
                                    vector4 := #EZ4,
                                    A_1 => #AA);
   "fuzzyfica"(crisp := #de,
                                    vector1 := #DEN1,
                                    vector2 := #DEN2,
                                    vector3 := #DEN3,
                                    vector4 := #DEN4,
                                    A_1 => #BB);
   #R4 := MIN_REAL(IN1 := #AA, IN2 := #BB);
   "fuzzyfica"(crisp := #e,
                                    vector1 := #EZ1,
                                    vector2 := #EZ2,
                                    vector3 := #EZ3,
                                    vector4 := #EZ4,
                                    A_1 => #AA);
   "fuzzyfica"(crisp := #de,
                                    vector1 := #DEZ1,
                                    vector2 := #DEZ2,
                                    vector3 := #DEZ3,
                                    vector4 := #DEZ4,
                                    A_1 => #BB);
   #R5 := MIN_REAL(IN1 := #AA, IN2 := #BB);
   "fuzzyfica"(crisp := #e,
                                    vector1 := #EZ1,
                                    vector2 := #EZ2,
                                    vector3 := #EZ3,
                                    vector4 := #EZ4,
                                    A_1 => #AA);
   "fuzzyfica"(crisp := #de,
                                    vector1 := #DEP1,
                                    vector2 := #DEP2,
                                    vector3 := #DEP3,
                                    vector4 := #DEP4,
                                    A_1 => #BB);
   #R6 := MIN_REAL(IN1 := #AA, IN2 := #BB);
   "fuzzyfica"(crisp := #e,
                                    vector1 := #EP1,
                                    vector2 := #EP2,
                                    vector3 := #EP3,
                                    vector4 := #EP4,
                                    A_1 => #AA);
   "fuzzyfica"(crisp := #de,
                                    vector1 := #DEZ1,
                                    vector2 := #DEZ2,
                                    vector3 := #DEZ3,
                                    vector4 := #DEZ4,
                                    A_1 => #BB);
   #R7 := MIN_REAL(IN1 := #AA, IN2 := #BB);
   "fuzzyfica"(crisp := #e,
                                    vector1 := #EP1,
                                    vector2 := #EP2,
                                    vector3 := #EP3,
                                    vector4 := #EP4,
                                    A_1 => #AA);
   "fuzzyfica"(crisp := #de,
                                    vector1 := #DEP1,
                                    vector2 := #DEP2,
                                    vector3 := #DEP3,
                                    vector4 := #DEP4,
                                    A_1 => #BB);
   #R8 := MIN_REAL(IN1 := #AA, IN2 := #BB);
   "fuzzyfica"(crisp := #e,
                                    vector1 := #EP1,
                                    vector2 := #EP2,
                                    vector3 := #EP3,
                                    vector4 := #EP4,
                                    A_1 => #AA);
   "fuzzyfica"(crisp := #de,
                                    vector1 := #DEN1,
                                    vector2 := #DEN2,
                                    vector3 := #DEN3,
                                    vector4 := #DEN4,
                                    A_1 => #BB);
   #R9 := MIN_REAL(IN1 := #AA, IN2 := #BB);
   #SS := ((#R1 * #N) + (#R2 * #N) + (#R3 * #Z) + (#R4 * #N) + (#R5 * #Z) + (#R6 * #P) + (#R7 * #P) + (#R8 * #P) + (#R9 * #P)) / (#R1 + #R2 + #R3 + #R4 + #R5 + #R6 + #R7 + #R8 + #R9);
   #S := (#var + #SS*1.3)+#pi;
END_FUNCTION_BLOCK

FUNCTION_BLOCK "smith"   // FB7, SCL
{ S7_Optimized_Access := 'TRUE' }
VERSION : 0.1
   VAR_INPUT
      ref : Real;
      refant : Real;
      kp : Real := 154.79;
      ki : Real := 1.083;
      sensorant : Real;
      sensor2ant : Real;
      kd : Real := 0.0;
      variador : Real;
      valprop : Real;
      sensor : Real;
   END_VAR
   VAR_OUTPUT
      u : Real;
      Scy : Real;
      Scy2ant : Real;
      Scyant : Real;
      Scrant : Real;
      Scr : Real;
      cont : Real;
      error : Real;
      e0 : Real;
      de : Real;
      contant : Real;
      "a" : Real;
      bant : Real;
      d : Real;
      c : Real;
      "b" : Real;
      aant : Real;
      ei : Real;
   END_VAR
BEGIN
   #Scr := (1.403*#ref)-(1.397*#refant)+ #Scrant;
   #u := #Scr- #Scy;
   #Scy := (2.932 * #sensor) - (5.857 * #sensorant) + (2.925 * #sensor2ant) + (1.999 * #Scyant) - (0.999 * #Scy2ant);

   #refant := #ref;
   #Scrant := #Scr;
   #sensor2ant := #sensorant;
   #sensorant := #sensor;
   #Scy2ant := #Scyant;
   #Scyant := #Scy;


   IF #u > 27000.0 THEN
       #u := 27000.0;
   END_IF;

   IF #u < 9000.0 THEN
       #u := 9000.0;
   END_IF;
END_FUNCTION_BLOCK

FUNCTION_BLOCK "smithanticipativo"   // FB8, SCL
{ S7_Optimized_Access := 'TRUE' }
VERSION : 0.1
   VAR_INPUT
      ref : Real;
      kp : Real := 154.79;
      ki : Real := 1.083;
      kd : Real := 0.0;
      variador : Real;
      valprop : Real;
      sensor : Real;
   END_VAR
   VAR_OUTPUT
      cont : Real;
      error : Real;
      e0 : Real;
      de : Real;
      contant : Real;
      "a" : Real;
      bant : Real;
      d : Real;
      c : Real;
      "b" : Real;
      aant : Real;
      k : Real;
      j : Real;
      hant : Real;
      h : Real;
      gant : Real;
      g : Real;
      jant : Real;
      kant : Real;
      iant : Real;
      l : Real;
      lant : Real;
      i : Real;
      varant : Real;
      ei : Real;
   END_VAR
BEGIN
   #error := #ref - #j;
   #ei := #ei + #error * 0.01;//periodo de muestreo t
   //#de := (#error - #e0) / 0.01;
   //7.2722 49.6172;
   #cont := (#kp * #error + #ki * #ei);
   #i := (#valprop*-0.002083) + (0.002047*#varant) + (0.9913*#iant);
   #iant := #i;
   #h := (-0.0006298*#i) + (#iant) + (0.0006298*#hant);
   #hant := #h;
   #g := #h + #cont;
   #a := (#g*0.000002235)+(#gant*0.000002235)+(#aant*0.98);
   #b := (#a*-0.9677)+(#aant)+(#bant*0.9677);
   #aant := #a;
   #bant := #b;
   #c:=#sensor-#b;
   #d:=#a+#c;

   (*#l := (#variador*0.000000465) + (#varant*0.000000465) + (0.9914*#lant);
   #lant := #l;
   #k := (-0.9952*#l) + (#lant) + (0.9952*#kant);
   #kant := #k;
   #gant := #g;*)
   #j := #d;
   #contant := #cont;
   #varant := #valprop;
   IF #cont > 27000.0 THEN
       #cont := 27000.0;
   END_IF;
   IF #cont < 9000.0 THEN
       #cont := 9000.0;
   END_IF;
END_FUNCTION_BLOCK

FUNCTION_BLOCK "lgr"   // FB9, SCL
{ S7_Optimized_Access := 'TRUE' }
VERSION : 0.1
   VAR_INPUT
      ref : Real;
      kp : Real := 0.0;
      ki : Real := 0.0;
      kd : Real := 0.0;
      refant : Real;
      sensorant : Real;
      sensor2ant : Real;
      sensor : Real;
   END_VAR
   VAR_OUTPUT
      señal_u : Real;
      Scrant : Real;
      Scyant : Real;
      Scy2ant : Real;
      Scy : Real;
      u : Real;
      Scr : Real;
      Scr2ant : Real;
      error2ant : Real;
      errorant : Real;
      error : Real;
      e0 : Real;
      de : Real;
      e1 : Real;
   END_VAR
BEGIN
   #error := #ref - #sensor;
   //#Scr := (1.4280 * #error) - (1.3623 * #errorant) + #Scrant;

   #Scr := (3071 * #error) - (6138 * #errorant) + (3068* #error2ant) + (1 * #Scr2ant);

   #refant := #ref;
   #Scrant := #Scr;
   #sensor2ant := #sensorant;
   #sensorant := #sensor;
   #Scr2ant := #Scrant;
   #Scrant := #Scy;
   #error2ant := #errorant;
   #errorant := #error;


   IF #Scr > 27000.0 THEN
       #Scr := 27000.0;
   END_IF;

   IF #Scr < 9000.0 THEN
       #Scr := 9000.0;
   END_IF;
END_FUNCTION_BLOCK

FUNCTION_BLOCK "controltemperatura"   // FB10, SCL
{ S7_Optimized_Access := 'TRUE' }
VERSION : 0.1
   VAR_INPUT
      temperatura : Real;
      setpoint : Real;
   END_VAR
   VAR_OUTPUT
      unidadcalentadora : Bool;
      unidadenfriadora : Bool;
   END_VAR
   VAR CONSTANT
      porcentaje : Real;
   END_VAR
BEGIN
   IF #temperatura> #setpoint THEN
       #unidadenfriadora :=1;
       #unidadcalentadora := 0;
   END_IF;
   IF #temperatura < #setpoint THEN
       #unidadenfriadora := 0;
       #unidadcalentadora := 1;
   END_IF;
END_FUNCTION_BLOCK

FUNCTION_BLOCK "OnOff_nivel"   // FB11, SCL
{ S7_Optimized_Access := 'TRUE' }
VERSION : 0.1
   VAR_INPUT
      setpoint : Real;
      sensor : Real;
   END_VAR
   VAR_OUTPUT
      vaciadoT1 : Bool;
      vaciadoT2 : Bool;
      llenadoT1 : Bool;
      llenadoT2 : Bool;
   END_VAR
BEGIN
   IF #sensor > #setpoint THEN
       #vaciadoT1 := 0;
       #vaciadoT2 := 1;
       #llenadoT1 := 1;
       #llenadoT2 := 0;
   END_IF;
   IF #sensor < #setpoint THEN
       #vaciadoT1 := 1;
       #vaciadoT2 := 0;
       #llenadoT1 := 0;
       #llenadoT2 := 1;
   END_IF;
END_FUNCTION_BLOCK

FUNCTION_BLOCK "OnOff_peso"   // FB12, SCL
{ S7_Optimized_Access := 'TRUE' }
VERSION : 0.1
   VAR_INPUT
      setpoint : Real;
      sensor : Real;
   END_VAR
   VAR_OUTPUT
      vaciadoT1 : Bool;
      vaciadoT2 : Bool;
      llenadoT1 : Bool;
      llenadoT2 : Bool;
   END_VAR
BEGIN
   IF #sensor > #setpoint THEN
       #vaciadoT1 := 1;
       #vaciadoT2 := 0;
       #llenadoT1 := 0;
       #llenadoT2 := 1;
   END_IF;
   IF #sensor < #setpoint THEN
       #vaciadoT1 := 0;
       #vaciadoT2 := 1;
       #llenadoT1 := 1;
       #llenadoT2 := 0;
   END_IF;
END_FUNCTION_BLOCK

FUNCTION_BLOCK "pid NIVEL"   // FB13, SCL
{ S7_Optimized_Access := 'TRUE' }
VERSION : 0.1
   VAR_INPUT
      ref : Real;
      kp : Real;
      ki : Real;
      kd : Real;
      sensor : Real;
   END_VAR
   VAR_OUTPUT
      señal_u : Real;
      VACIADOT1 : Bool;
      VACIADOT2 : Bool;
      LLENADOT2 : Bool;
      LLENADOT1 : Bool;
      error : Real;
      e1 : Real;
      de : Real;
      e0 : Real;
   END_VAR
BEGIN
   #error := #ref - #sensor;
   #e1 := #e1 + #error * 0.01;//periodo de muestreo t
   #de := (#error - #e0) / 0.01;
   #señal_u := (#kp * #error + #ki * #e1 + #de * #kd);
   IF #error > 0 THEN
       #VACIADOT1 := 1;
       #VACIADOT2 := 0;
       #LLENADOT1 := 0;
       #LLENADOT2 := 1;
   ELSE
       #VACIADOT1 := 0;
       #VACIADOT2 := 1;
       #LLENADOT1 := 1;
       #LLENADOT2 := 0;
   END_IF;

   IF #señal_u > 27000.0 THEN
       #señal_u := 27000.0;
   END_IF;
   IF #señal_u < 9000.0 THEN
       #señal_u := 9000.0;
   END_IF;
END_FUNCTION_BLOCK

FUNCTION_BLOCK "PID_FLUJO"   // FB14, SCL
{ S7_Optimized_Access := 'TRUE' }
VERSION : 0.1
   VAR_INPUT
      ref : Real;
      sensor : Real;
      rdisturbance : Real;
   END_VAR
   VAR_OUTPUT
      Motor : Real;
      Ojo : Real;
   END_VAR
   VAR_TEMP
      "e" : Real;
      de : Real;
      ie : Real;
      e3 : Real;
      e1 : Real;
      Bomba : Real;
      uc2 : Real;
      u : Real;
      u1 : Real;
      u2 : Real;
      baux : Real;
      e2 : Real;
      ud : Real;
      uc : Real;
      ds : Real;
      uaux : Real;
      eaux : Real;
   END_VAR
   VAR CONSTANT
      ecn : Real := 244.0784;
      ecn1 : Real := 892.0721;
      ecn2 : Real := 1221.698;
      ecn3 : Real := 742.9892;
      ecn4 : Real := 169.2944;
      ucn1 : Real := 3.2507;
      ucn2 : Real := 3.8764;
      ucn3 : Real := 1.9963;
      err2 : Real := 0.0;
      Constant_3 : Real;
      Constant_1 : Real;
      Constant_2 : Real;
      ucn4 : Real := 0.3706;
   END_VAR
BEGIN
   #e := #ref - #sensor;
   //#ds :=27000-  #rdisturbance;
   #Ojo := #e;
   //#u := (#ecn * #e) - (#ecn1 * "PresionZd".e1) + (#ecn2 * "PresionZd".e2) - (#ecn3 * "PresionZd".e3) + (#ecn4 * "PresionZd".e4)
   //+ (#ucn1 * "PresionZd".u1) - (#ucn2 * "PresionZd".u2) + (#ucn3 * "PresionZd".u3) - (#ucn4 * "PresionZd".u4);


   //#ud := 0.2271* #ds -0.4558* "PresionZd".ds1 +0.2281* "PresionZd".ds2
   //+1.909* "PresionZd".ud1 -0.9114*"PresionZd".ud2;
   //
   //#u := (#ecn * #e) - (#ecn1 * "PresionZd".e1) + (#ecn2 * "PresionZd".e2) - (#ecn3 * "PresionZd".e3) + (#ecn4 * "PresionZd".e4)
   //+ (#ucn1 * "PresionZd".u1) - (#ucn2 * "PresionZd".u2) + (#ucn3 * "PresionZd".u3) - (#ucn4 * "PresionZd".u4);
   #u := 148.1*#e-263.9*#e1+117.8*#e2+1.868*#uc-0.8684*#uc2;
   //#u := 76.31 * #e - 143.2 * #e1 + 67.44 * #e2 + 1.874 * #uc - 0.874 * #uc2;

   #uaux := #uc;
   #uc := #u;
   #uc2 := #uaux;

   #baux := #u;//
   #eaux := #e1;
   #e1 := #e;
   #e2 := #eaux;


   IF #baux > 27000.0 THEN
       #Motor := 27000.0;
   ELSIF #baux < 6500.0 THEN
       #Motor := 6500.0;
   ELSE
       #Motor := #baux;
   END_IF;


   //"PresionZd".e4 := "PresionZd".e3;
   //"PresionZd".e3 := "PresionZd".e2;
   //"PresionZd".e2 := "PresionZd".e1;
   //"PresionZd".e1 := #e;

   //"PresionZd".u4 := "PresionZd".u3;
   //"PresionZd".u3 := "PresionZd".u2;
   //"PresionZd".u2 := "PresionZd".u1;
   //"PresionZd".u1 := #u;

   //"PresionZd".ds2 := "PresionZd".ds1;
   //"PresionZd".ds1 := #ds;

   //"PresionZd".ud2 := "PresionZd".ud1;
   //"PresionZd".ud1 := #ud;
END_FUNCTION_BLOCK

FUNCTION_BLOCK "Bloque_2"   // FB15, SCL
{ S7_Optimized_Access := 'TRUE' }
VERSION : 0.1
   VAR_INPUT
      sp : Real;
      y : Real;
      kp : Real;
      ti : Real;
      td : Real;
   END_VAR
   VAR_OUTPUT
      "M" : Real;
   END_VAR
   VAR
      e0 : Real := 0.0;
      e1 : Real;
      de : Real;
      ie : Real;
      ki : Real;
      kd : Real;
   END_VAR
BEGIN
   #e1:=#sp - #y;
   #de := (#e1 - #e0) /  0.01;
   #ie := #ie + (#e1 *  0.01);
   #ki := #kp / #ti;
   #kd:= #kp * #td;
   #M:= #e1*#kp + #ie*#ki +#de*#kd;
   IF #M>32000 THEN
       // Statement section IF
       #M :=32000;
   END_IF;
   IF #M<6500 THEN
       // Statement section IF
       #M := 6500;
   END_IF;

   #e0:=#e1;
END_FUNCTION_BLOCK

FUNCTION_BLOCK "Caracterizacion"   // FB16, LAD
{ S7_Optimized_Access := 'TRUE' }
VERSION : 0.1
   VAR_INPUT
      inicio_llenadot1 : Bool;
      valor_variador : Int;
      valor_valvula : Int;
      inicio_presion : Bool;
      inicio_llenadot2 : Bool;
      inicio_flujo : Bool;
      inicio_temp : Bool;
   END_VAR
   VAR_OUTPUT
      onoff_variador : Bool;
      valv1 : Bool;
      valv2 : Bool;
      valv_pro : Int;
      vaciadot2 : Bool;
      calentador : Bool;
      vaciadot1 : Bool;
   END_VAR
BEGIN

REGION Network 1: medición de nivel tanque 2
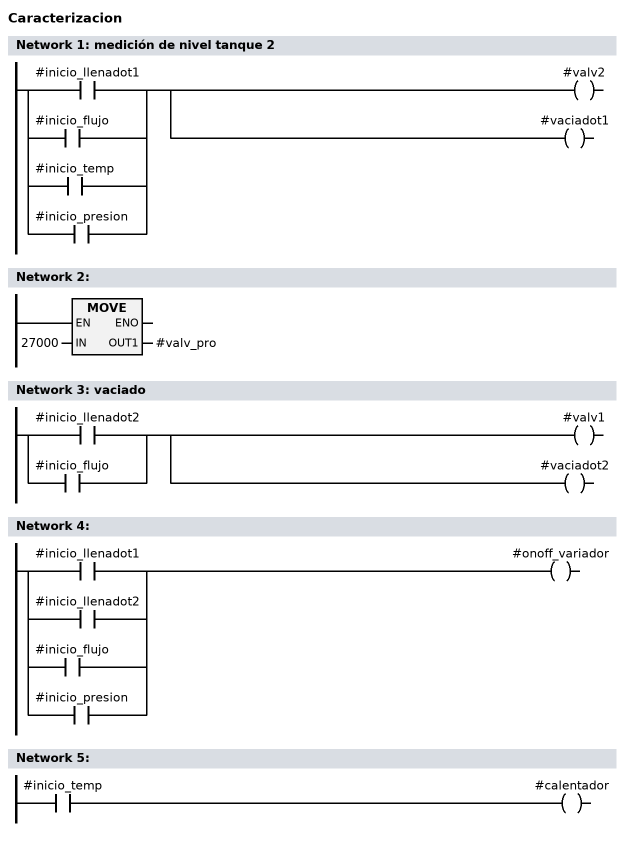
   RUNG wire#powerrail
      Contact( #inicio_llenadot1 )
      wire#w1
      Coil( #valv2 )
   END_RUNG
   RUNG wire#powerrail
      Contact( #inicio_flujo )
   END_RUNG wire#w1
   RUNG wire#powerrail
      Contact( #inicio_temp )
   END_RUNG wire#w1
   RUNG wire#powerrail
      Contact( #inicio_presion )
   END_RUNG wire#w1
   RUNG wire#w1
      Coil( #vaciadot1 )
   END_RUNG
   // the same network as SCL:
   #valv2 := #inicio_llenadot1 OR #inicio_flujo OR #inicio_temp OR #inicio_presion;
   #vaciadot1 := #valv2;
END_REGION

REGION Network 2
   RUNG wire#powerrail
      Move(in := 27000, out1 => #valv_pro)
   END_RUNG
   // the same network as SCL:
   #valv_pro := 27000;
END_REGION

REGION Network 3: vaciado
   RUNG wire#powerrail
      Contact( #inicio_llenadot2 )
      wire#w1
      Coil( #valv1 )
   END_RUNG
   RUNG wire#powerrail
      Contact( #inicio_flujo )
   END_RUNG wire#w1
   RUNG wire#w1
      Coil( #vaciadot2 )
   END_RUNG
   // the same network as SCL:
   #valv1 := #inicio_llenadot2 OR #inicio_flujo;
   #vaciadot2 := #valv1;
END_REGION

REGION Network 4
   RUNG wire#powerrail
      Contact( #inicio_llenadot1 )
      wire#w1
      Coil( #onoff_variador )
   END_RUNG
   RUNG wire#powerrail
      Contact( #inicio_llenadot2 )
   END_RUNG wire#w1
   RUNG wire#powerrail
      Contact( #inicio_flujo )
   END_RUNG wire#w1
   RUNG wire#powerrail
      Contact( #inicio_presion )
   END_RUNG wire#w1
   // the same network as SCL:
   #onoff_variador := #inicio_llenadot1 OR #inicio_llenadot2 OR #inicio_flujo OR #inicio_presion;
END_REGION

REGION Network 5
   RUNG wire#powerrail
      Contact( #inicio_temp )
      Coil( #calentador )
   END_RUNG
   // the same network as SCL:
   #calentador := #inicio_temp;
END_REGION
END_FUNCTION_BLOCK

FUNCTION_BLOCK "Calibracion_Nivel"   // FB17, LAD
{ S7_Optimized_Access := 'TRUE' }
VERSION : 0.1
   VAR_INPUT
      nivTanq : Int;
   END_VAR
   VAR_OUTPUT
      "Ax+B" : Real;
   END_VAR
   VAR
      Ax : Real;
      Static_1 : Real;
   END_VAR
BEGIN

REGION Network 1
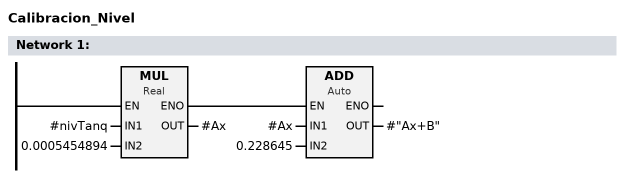
   RUNG wire#powerrail
      { S7_Templates := "SrcType := Real" } Mul(in1 := #nivTanq, in2 := 0.0005454894, out => #Ax)
      Add(in1 := #Ax, in2 := 0.228645, out => #"Ax+B")
   END_RUNG
   // the same network as SCL:
   #Ax := #nivTanq * 0.0005454894;
   #"Ax+B" := #Ax + 0.228645;
END_REGION
END_FUNCTION_BLOCK

FUNCTION_BLOCK "Calibracion Presion"   // FB18, LAD
{ S7_Optimized_Access := 'TRUE' }
VERSION : 0.1
   VAR_INPUT
      presion : Real;
   END_VAR
   VAR_OUTPUT
      "Ax-B" : Real;
   END_VAR
   VAR
      Ax : Real;
   END_VAR
BEGIN

REGION Network 1
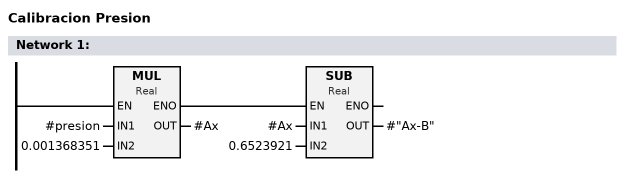
   RUNG wire#powerrail
      { S7_Templates := "SrcType := Real" } Mul(in1 := #presion, in2 := 0.001368351, out => #Ax)
      { S7_Templates := "SrcType := Real" } Sub(in1 := #Ax, in2 := 0.6523921, out => #"Ax-B")
   END_RUNG
   // the same network as SCL:
   #Ax := #presion * 0.001368351;
   #"Ax-B" := #Ax - 0.6523921;
END_REGION
END_FUNCTION_BLOCK

FUNCTION_BLOCK "Calibracion temperatura"   // FB19, LAD
{ S7_Optimized_Access := 'TRUE' }
VERSION : 0.1
   VAR_INPUT
      Temperaturaa : Real;
   END_VAR
   VAR_OUTPUT
      "Ax-B" : Real;
   END_VAR
   VAR
      Ax : Real;
   END_VAR
BEGIN

REGION Network 1
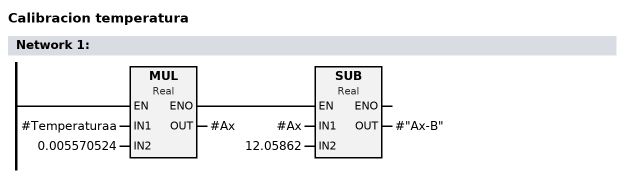
   RUNG wire#powerrail
      { S7_Templates := "SrcType := Real" } Mul(in1 := #Temperaturaa, in2 := 0.005570524, out => #Ax)
      { S7_Templates := "SrcType := Real" } Sub(in1 := #Ax, in2 := 12.05862, out => #"Ax-B")
   END_RUNG
   // the same network as SCL:
   #Ax := #Temperaturaa * 0.005570524;
   #"Ax-B" := #Ax - 12.05862;
END_REGION
END_FUNCTION_BLOCK

FUNCTION_BLOCK "Calibracion Flujo"   // FB20, LAD
{ S7_Optimized_Access := 'TRUE' }
VERSION : 0.1
   VAR_INPUT
      flujo : Real;
   END_VAR
   VAR_OUTPUT
      "Ax-B" : Real;
   END_VAR
   VAR
      Ax : Real;
   END_VAR
BEGIN

REGION Network 1
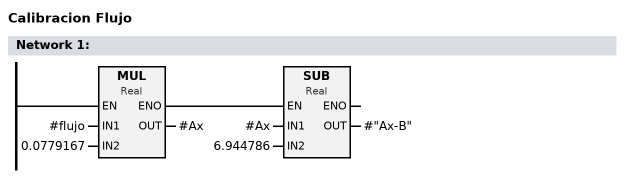
   RUNG wire#powerrail
      { S7_Templates := "SrcType := Real" } Mul(in1 := #flujo, in2 := 0.0779167, out => #Ax)
      { S7_Templates := "SrcType := Real" } Sub(in1 := #Ax, in2 := 6.944786, out => #"Ax-B")
   END_RUNG
   // the same network as SCL:
   #Ax := #flujo * 0.0779167;
   #"Ax-B" := #Ax - 6.944786;
END_REGION
END_FUNCTION_BLOCK

FUNCTION_BLOCK "PID_PRESION"   // FB21, SCL
{ S7_Optimized_Access := 'TRUE' }
VERSION : 0.1
   VAR_INPUT
      ref : Real;
      sensor : Real;
      rdisturbac : Word;
   END_VAR
   VAR_OUTPUT
      Motor : Real;
   END_VAR
   VAR_TEMP
      "e" : Real;
      de : Real;
      ie : Real;
      e1 : Real;
      Bomba : Real;
      u : Real;
      u1 : Real;
      u2 : Real;
      uc : Real;
      ud : Real;
      baux : Real;
      e2 : Real;
      ds : Real;
   END_VAR
   VAR CONSTANT
      ecn : Real := 848.2595;
      ecn1 : Real := 2084.463;
      ecn2 : Real := 1898.801;
      ecn3 : Real := 758.3437;
      ecn4 : Real := 111.7074;
      ucn1 : Real := 2.9557;
      ucn2 : Real := 3.2566;
      ucn3 : Real := 1.5588;
      ucn4 : Real := 0.2797;
   END_VAR
BEGIN
   #e := #ref - #sensor;
   #ds := 27000-#rdisturbac;

   #u := (#ecn*#e) -(#ecn1*"PresionZd".e1) +(#ecn2*"PresionZd".e2) -(#ecn3*"PresionZd".e3) +(#ecn4*"PresionZd".e4)
   +(#ucn1 *"PresionZd".u1) -(#ucn2*"PresionZd".u2) +(#ucn3*"PresionZd".u3) -(#ucn4*"PresionZd".u4);


   #ud:=42.17 *#ds - 98.43 *"PresionZd".ds1+ 2.976*"PresionZd".ds2
   +0.03197*"PresionZd".ud1 -4.495e-09*"PresionZd".ud2;

   #uc := #u + #ud;
   #baux := #uc; 

   IF #baux > 27000.0 THEN
       #Motor := 27000.0;
   ELSIF #baux < 6500.0 THEN
       #Motor := 6500.0;
   ELSE
       #Motor := #baux;
   END_IF;


   "PresionZd".e4 := "PresionZd".e3;
   "PresionZd".e3 := "PresionZd".e2;
   "PresionZd".e2 := "PresionZd".e1;
   "PresionZd".e1 := #e;

   "PresionZd".u4 := "PresionZd".u3;
   "PresionZd".u3 := "PresionZd".u2;
   "PresionZd".u2 := "PresionZd".u1;
   "PresionZd".u1 := #u;

   "PresionZd".ds2:="PresionZd".ds1;
   "PresionZd".ds1 := #ds;

   "PresionZd".ud2 := "PresionZd".ud1;
   "PresionZd".ud1 := #ud;
END_FUNCTION_BLOCK

FUNCTION_BLOCK "smith completo"   // FB22, SCL
{ S7_Optimized_Access := 'TRUE' }
VERSION : 0.1
   VAR_INPUT
      setpoint : Real;
      sensor : Real;
   END_VAR
   VAR_OUTPUT
      bomba : Real;
      VACIADOT1 : Bool;
      VACIADOT2 : Bool;
      LLENADOT1 : Bool;
      LLENADOT2 : Bool;
   END_VAR
   VAR_TEMP
      "e" : Real;
      e1 : Real;
      e2 : Real;
      u1 : Real;
      u2 : Real;
      y1 : Real;
      y11 : Real;
      y12 : Real;
      y2 : Real;
      y21 : Real;
      y22 : Real;
      y23 : Real;
      y3 : Real;
      y4 : Real;
   END_VAR
BEGIN
   #e :=  #setpoint-#y4;


   //#bomba := (16.73  * #e) - (33.45 * #e1) + (16.73 * #e2) + #u2;
   #bomba := (0.02946* #e) - (0.02944* #e1)  + #u1;
   //16.73
   //33.45
   //16.73

   #y1 :=#y11  + 0.0002316 * #u1;


   #y2 := -#y1 + #y11 + 0.9037* #y21;


   IF #bomba > 27000.0 THEN
       #bomba := 27000.0;
   END_IF;
   IF #bomba < 9000.0 THEN
       #bomba := 9000.0;
   END_IF;
   #u1 := #bomba;
   #e1 := #e;

   #y3 := #sensor - #y2;
   #y4 := #y1 + #y3;
   #y11 := #y1;
   #y12 := #y11;
   #y21 := #y2;

   #e2 := #e1;
END_FUNCTION_BLOCK

FUNCTION_BLOCK "Smith_please"   // FB23, SCL
{ S7_Optimized_Access := 'TRUE' }
VERSION : 0.1
   VAR_INPUT
      Sensor : Real;
      Ref : Real;
   END_VAR
   VAR_OUTPUT
      Bomba : Real;
   END_VAR
   VAR_TEMP
      "e" : Real;
      u1 : Real;
      e1 : Real;
      y4 : Real;
      y1 : Real;
      y3 : Real;
      y11 : Real;
      y2 : Real;
      y21 : Real;
      aux : Real;
   END_VAR
BEGIN


   #y3 := #Sensor - #y2;
   #y4 := #y1 + #y3;
   #e := #Ref - #y4;


   //#bomba := (16.73  * #e) - (33.45 * #e1) + (16.73 * #e2) + #u2;
   #aux := (0.02946 * #e) - (0.02944 * #e1) + #u1;

   IF #aux > 27000.0 THEN
       #Bomba := 27000.0;
   ELSIF #aux < 9000.0 THEN
       #Bomba := 9000.0;
   ELSE
       #Bomba := #aux;
   END_IF;


   #e1 := #e;
   #u1 := #aux;


   #y2 := - #y1 + #y11 + (0.9997 * #y21);
   #y1 := #y11 + (2316 * #u1);
   #y11 := #y1;
   #y21 := #y2;
END_FUNCTION_BLOCK

FUNCTION_BLOCK "CALCULO_FLUJO"   // FB24, LAD
{ S7_Optimized_Access := 'TRUE' }
VERSION : 0.1
   VAR_INPUT
      Nivel : Real;
      plcflujo : Real;
   END_VAR
   VAR_OUTPUT
      Flujo : Real;
   END_VAR
   VAR
      T1 : IEC_TIMER;
      C1 : IEC_COUNTER;
   END_VAR
   VAR RETAIN
      T2 : IEC_TIMER;
   END_VAR
   VAR
      T3 : IEC_TIMER;
      T4 : IEC_TIMER;
      T5 : IEC_TIMER;
      T6 : IEC_TIMER;
      T7 : IEC_TIMER;
      CONTEO : Int;
      Flujo2 : Real;
   END_VAR
   VAR_TEMP
      DELTA : Real;
      deltan1 : Real;
      deltan2 : Real;
   END_VAR
BEGIN

REGION Network 1
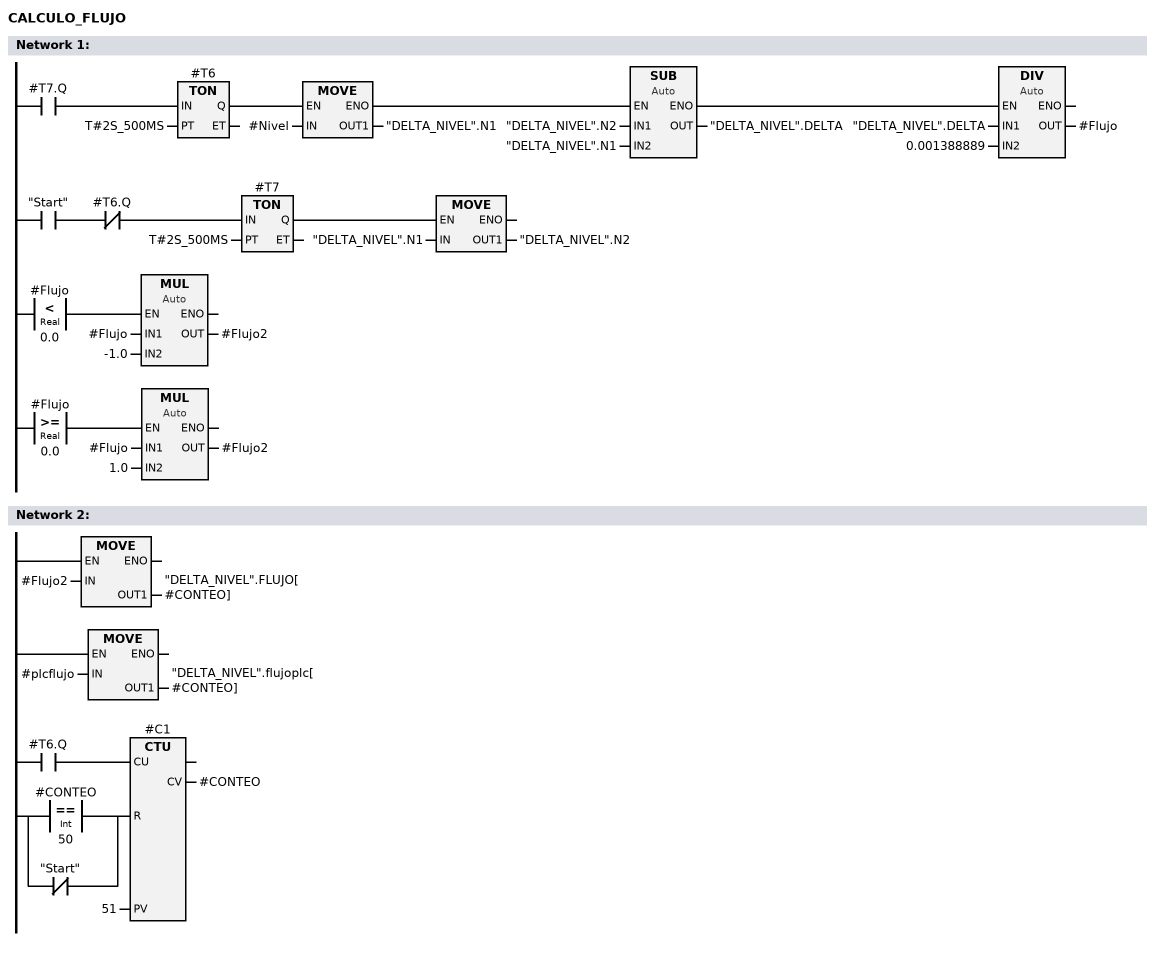
   #T6.TON(IN := #T7.Q, PT := T#2S_500MS);
   IF #T6.Q THEN
       "DELTA_NIVEL".N1 := #Nivel;
       "DELTA_NIVEL".DELTA := "DELTA_NIVEL".N2 - "DELTA_NIVEL".N1;
       #Flujo := "DELTA_NIVEL".DELTA / 0.001388889;
   END_IF;
   #T7.TON(IN := "Start" AND NOT #T6.Q, PT := T#2S_500MS);
   IF #T7.Q THEN "DELTA_NIVEL".N2 := "DELTA_NIVEL".N1; END_IF;
   IF #Flujo < 0.0 THEN #Flujo2 := #Flujo * (-1.0); END_IF;
   IF #Flujo >= 0.0 THEN #Flujo2 := #Flujo * 1.0; END_IF;
END_REGION

REGION Network 2
   "DELTA_NIVEL".FLUJO[#CONTEO] := #Flujo2;
   "DELTA_NIVEL".flujoplc[#CONTEO] := #plcflujo;
   #C1.CTU(CU := #T6.Q, R := (#CONTEO = 50) OR NOT "Start", PV := 51, CV => #CONTEO);
END_REGION
END_FUNCTION_BLOCK

FUNCTION_BLOCK "PID_JyH"   // FB25, SCL
{ S7_Optimized_Access := 'TRUE' }
VERSION : 0.1
   VAR_INPUT
      ref : Real;
      u1_in : Real;
      u2_in : Real;
      e1_in : Real;
      e2_in : Real;
      flujo : Real;
   END_VAR
   VAR_OUTPUT
      u1_out_1 : Real;
      u2_out_1 : Real;
      e1_out_1 : Real;
      e2_out_1 : Real;
      Motor : Real;
   END_VAR
   VAR_TEMP
      u : Real;
      u1 : Real;
      u2 : Real;
      "e" : Real;
      e1 : Real;
      e2 : Real;
      baux : Real;
      auxbomba : Real;
   END_VAR
BEGIN
   #e := #ref - #flujo;
   #e1 := #e1_in;
   #e2 := #e2_in;
   #u1 := #u1_in;
   #u2 := #u2_in;
   #u := 148.1 * #e - 263.9 * #e1 + 117.8 * #e2 + 1.868 * #u1 - 0.8684 * #u2;
   #baux := #u;

   IF #baux > 27000.0 THEN
       #Motor := 27000.0;
   ELSIF #baux < 6500.0 THEN
       #Motor := 6500.0;
   ELSE
       #Motor := #baux;
   END_IF;
   #e2 := #e1;
   #e2_out_1 := #e2;
   #e1 := #e;
   #e1_out_1 := #e;
   #u2 := #u1;
   #u2_out_1 := #u2;
   #u1 := #u;
   #u1_out_1 := #u1;
   #baux := #u;
END_FUNCTION_BLOCK

FUNCTION_BLOCK "Smith Flujo"   // FB26, SCL
{ S7_Optimized_Access := 'TRUE' }
VERSION : 0.1
   VAR_INPUT
      ref : Real;
      u1_in : Real;
      u2_in : Real;
      u3_in : Real;
      u4_in : Real;
      e1_in : Real;
      e2_in : Real;
      e3_in : Real;
      e4_in : Real;
      flujo : Real;
   END_VAR
   VAR_OUTPUT
      u1_out_1 : Real;
      u2_out_1 : Real;
      u3_out_1 : Real;
      u4_out_1 : Real;
      e1_out_1 : Real;
      e2_out_1 : Real;
      e3_out_1 : Real;
      e4_out_1 : Real;
      Motor : Real;
   END_VAR
   VAR_TEMP
      u : Real;
      u1 : Real;
      u2 : Real;
      u3 : Real;
      u4 : Real;
      "e" : Real;
      e0 : Real;
      e1 : Real;
      e2 : Real;
      e3 : Real;
      e4 : Real;
      baux : Real;
      auxbomba : Real;
   END_VAR
BEGIN

   #e := #ref - #flujo;

   #e1 := #e1_in;
   #e2 := #e2_in;
   #e3 := #e3_in;
   #e4 := #e4_in;

   #u1 := #u1_in;
   #u2 := #u2_in;
   #u3 := #u3_in;
   #u4 := #u4_in;

   // 44.0301 -171.1812  249.5333 -161.6410   39.2588
   // 1.0000no se toma u   -3.8658    5.6010   -3.6047    0.8694
   #u := 44.0301*#e - 171.1812*#e1 + 249.5333*#e2 -161.6410*#e3 +39.2588*#e4 + 3.8658*#u1 - 5.6010*#u2 +3.6047*#u3-0.8694*#u4;
   #baux := #u;

   IF #baux > 27000.0 THEN
       #Motor := 27000.0;
   ELSIF #baux < 6500.0 THEN
       #Motor := 6500.0;
   ELSE
       #Motor := #baux;
   END_IF;

   #e4 := #e3;
   #e3 := #e2;
   #e2 := #e1;
   #e1 := #e;

   #e4_out_1 := #e4;
   #e3_out_1 := #e3;
   #e2_out_1 := #e2;
   #e1_out_1 := #e;

   #u4 := #u3;
   #u3 := #u2;
   #u2 := #u1;
   #u1 := #baux;
   #u4_out_1 := #u4;
   #u3_out_1 := #u3;
   #u2_out_1 := #u2;
   #u1_out_1 := #u1;

   #baux := #u;
END_FUNCTION_BLOCK

FUNCTION_BLOCK "Smith Presion"   // FB27, SCL
{ S7_Optimized_Access := 'TRUE' }
VERSION : 0.1
   VAR_INPUT
      ref : Real;
      u1_in : Real;
      u2_in : Real;
      u3_in : Real;
      u4_in : Real;
      e1_in : Real;
      e2_in : Real;
      e3_in : Real;
      e4_in : Real;
      flujo : Real;
   END_VAR
   VAR_OUTPUT
      u1_out_1 : Real;
      u2_out_1 : Real;
      u3_out_1 : Real;
      u4_out_1 : Real;
      e1_out_1 : Real;
      e2_out_1 : Real;
      e3_out_1 : Real;
      e4_out_1 : Real;
      Motor : Real;
   END_VAR
   VAR_TEMP
      u : Real;
      u1 : Real;
      u2 : Real;
      u3 : Real;
      u4 : Real;
      "e" : Real;
      e0 : Real;
      e1 : Real;
      e2 : Real;
      e3 : Real;
      e4 : Real;
      baux : Real;
      auxbomba : Real;
   END_VAR
BEGIN
   #e := #ref - #flujo;
   #e1 := #e1_in;
   #e2 := #e2_in;
   #e3 := #e3_in;
   #e4 := #e4_in;

   #u1 := #u1_in;
   #u2 := #u2_in;
   #u3 := #u3_in;
   #u4 := #u4_in;

   //44.0301 -171.1812  249.5333 -161.6410   39.2588
   // 1.0000   -3.8658    5.6010   -3.6047    0.8694
   #u := 44.0301*#e - 171.1812*#e1 + 249.5333*#e2 -161.641*#e3 + 39.2588*#e4+3.8658*#u1 - 5.601*#u2 +3.6047*#u3-0.8694*#u4;
   #baux := #u;

   IF #baux > 27000.0 THEN
       #Motor := 27000.0;
   ELSIF #baux < 6500.0 THEN
       #Motor := 6500.0;
   ELSE
       #Motor := #baux;
   END_IF;

   #e4 := #e3;
   #e3 := #e2;
   #e2 := #e1;
   #e1 := #e;

   #e4_out_1 := #e4;
   #e3_out_1 := #e3;
   #e2_out_1 := #e2;
   #e1_out_1 := #e;

   #u4 := #u3;
   #u3 := #u2;
   #u2 := #u1;
   #u1 := #Motor;
   #u4_out_1 := #u4;
   #u3_out_1 := #u3;
   #u2_out_1 := #u2;
   #u1_out_1 := #u1;

   #baux := #u;
END_FUNCTION_BLOCK

FUNCTION_BLOCK "smith_flujo_definitivo"   // FB28, SCL
{ S7_Optimized_Access := 'TRUE' }
VERSION : 0.1
   VAR_INPUT
      ref : Real;
      u1_in : Real;
      u2_in : Real;
      u3_in : Real;
      u4_in : Real;
      e1_in : Real;
      e2_in : Real;
      e3_in : Real;
      e4_in : Real;
      flujo : Real;
   END_VAR
   VAR_OUTPUT
      u1_out_1 : Real;
      u2_out_1 : Real;
      u3_out_1 : Real;
      u4_out_1 : Real;
      e1_out_1 : Real;
      e2_out_1 : Real;
      e3_out_1 : Real;
      e4_out_1 : Real;
      Motor : Real;
   END_VAR
   VAR_TEMP
      u : Real;
      u1 : Real;
      u2 : Real;
      u3 : Real;
      u4 : Real;
      "e" : Real;
      e0 : Real;
      e1 : Real;
      e2 : Real;
      e3 : Real;
      e4 : Real;
      baux : Real;
      auxbomba : Real;
   END_VAR
BEGIN
   #e := #ref - #flujo;
   #e1 := #e1_in;
   #e2 := #e2_in;
   #e3 := #e3_in;
   #e4 := #e4_in;

   #u1 := #u1_in;
   #u2 := #u2_in;
   #u3 := #u3_in;
   #u4 := #u4_in;


   //Diseno Rodrizo
   //34.3535 -120.8427 159.3149 -93.2974 20.4776
   //1.000 -3.4148 4.3335 -2.4187 0.5
   //
   //#u := 34.3535 * #e- 120.842*#e1 + 159.3149* #e2 -93.2974* #e3 + 20.4776*#e4 + 3.4148*#u1 - 4.3335*#u2 + 2.4187*#u3-0.5*#u4;
   //diseno Juanito 
   // 8.1641  -22.2490   21.9482   -9.2391    1.4002
   // 1.0000   -3.1515    3.6052   -1.7482    0.2945
   // 
   //#u := 8.1641*#e-22.2490*#e1+21.9482*#e2-9.2391*#e3+1.4002*#e4+3.1515*#u1-3.6052*#u2+1.7482*#u3-0.2945*#u4;
   //NGcz =

   //5.7927  -15.3991   14.5405   -5.6418    0.7252
   //DGcz =
   //1.0000   -3.0322    3.2652   -1.4255    0.1925
   #u := 5.7927*#e -15.3991*#e1 + 14.5405* #e2 -5.6418*#e3 + 0.7252*#e4 + 3.0322*#u1-3.2652*#u2 +1.4255*#u3-0.1925* #u4;
   #baux := #u;

   IF #baux > 27000.0 THEN
       #Motor := 27000.0;
   ELSIF #baux < 6500.0 THEN
       #Motor := 6500.0;
   ELSE
       #Motor := #baux;
   END_IF;

   #e4 := #e3;
   #e3 := #e2;
   #e2 := #e1;
   #e1 := #e;

   #e4_out_1 := #e4;
   #e3_out_1 := #e3;
   #e2_out_1 := #e2;
   #e1_out_1 := #e;

   #u4 := #u3;
   #u3 := #u2;
   #u2 := #u1;
   #u1 := #baux;
   #u4_out_1 := #u4;
   #u3_out_1 := #u3;
   #u2_out_1 := #u2;
   #u1_out_1 := #u1;
END_FUNCTION_BLOCK

FUNCTION_BLOCK "filto"   // FB29, SCL
{ S7_Optimized_Access := 'TRUE' }
VERSION : 0.1
   VAR_INPUT
      presion : Real;
      e1_in : Real;
      e2_in : Real;
      u1_in : Real;
      u2_in : Real;
   END_VAR
   VAR_OUTPUT
      presion_filtrada : Real;
      e1_out_1 : Real;
      e2_out_2 : Real;
      u1_out_2 : Real;
      u2_out_1 : Real;
   END_VAR
   VAR_TEMP
      "e" : Real;
      e1 : Real;
      e2 : Real;
      u : Real;
      u1 : Real;
      u2 : Real;
   END_VAR
BEGIN
   //#presion
   //
   #e := #presion;
   #e1 := #e1_in;
   #e2 := #e2_in;

   #u1 := #u1_in;
   #u2 := #u2_in;


   // e 0.4574    0.9149    0.4574
   // u 1.0000    0.5949    0.2348
   #u := 0.4574*#e+0.9149*#e1 + 0.4574*#e2-0.5949*#u1-0.2348*#u2;//sirve
   //#u := 0.0055 * #e + 0.0111 * #e1 + 0.0055 * #e2 + 1.7786 * #u1 - 0.8008 * #u2;
   //#u := 0.0675 * #e + 0.1349* #e1 + 0.0675 * #e2 + 1.1430* #u1 - 0.4128*#u2;
   //corrimiento entrada
   #e2 := #e1;
   #e1 := #e;

   #e2_out_2 := #e2;
   #e1_out_1 := #e;

   #u2 := #u1;
   #u1 := #u;

   #u2_out_1 := #u2;
   #u1_out_2 := #u1;

   #presion_filtrada := #u;
END_FUNCTION_BLOCK

FUNCTION_BLOCK "smith_presion_definitivo"   // FB30, SCL
{ S7_Optimized_Access := 'TRUE' }
VERSION : 0.1
   VAR_INPUT
      ref : Real;
      u1_in : Real;
      u2_in : Real;
      u3_in : Real;
      u4_in : Real;
      e1_in : Real;
      e2_in : Real;
      e3_in : Real;
      e4_in : Real;
      flujo : Real;
   END_VAR
   VAR_OUTPUT
      u1_out_1 : Real;
      u2_out_1 : Real;
      u3_out_1 : Real;
      u4_out_1 : Real;
      e1_out_1 : Real;
      e2_out_1 : Real;
      e3_out_1 : Real;
      e4_out_1 : Real;
      Motor : Real;
   END_VAR
   VAR_TEMP
      u : Real;
      u1 : Real;
      u2 : Real;
      u3 : Real;
      u4 : Real;
      "e" : Real;
      e0 : Real;
      e1 : Real;
      e2 : Real;
      e3 : Real;
      e4 : Real;
      baux : Real;
      auxbomba : Real;
   END_VAR
BEGIN
   #e := #ref - #flujo;
   #e1 := #e1_in;
   #e2 := #e2_in;
   #e3 := #e3_in;
   #e4 := #e4_in;

   #u1 := #u1_in;
   #u2 := #u2_in;
   #u3 := #u3_in;
   #u4 := #u4_in;

   // 8.1641  -22.2490   21.9482   -9.2391    1.4002
   // 1.0000   -3.1515    3.6052   -1.7482    0.2945
   // 
   //#u := 8.1641*#e-22.2490*#e1+21.9482*#e2-9.2391*#e3+1.4002*#e4+3.1515*#u1-3.6052*#u2+1.7482*#u3-0.2945*#u4;
   //1.0e+03 *
   //2.3516   -5.9254    5.3604   -2.0103    0.2482
   //1.0000   -3.1401    3.6865   -1.9253    0.3789

   //Funcionando
   //#u := 2351.6*#e-5925.4*#e1+5360.4*#e2 -2010.3* #e3 +  248.2*#e4 + 3.1401*#u1-3.6865*#u2+1.9253*#u3-0.3789*#u4;
   // *1000 1.8644   -4.0330    3.0455   -0.9306    0.0968
   //1.0000   -2.8751    2.9996   -1.3355    0.2110
   //
   #u := 1864.4 * #e - 4033.0 * #e1 + 3045.5 * #e2 - 930.6 * #e3 + 96.8 * #e4 + 2.8751 * #u1 - 2.9996 * #u2 + 1.3355 * #u3 - 0.2110 * #u4;
   #baux := #u;

   IF #baux > 27000.0 THEN
       #Motor := 27000.0;
   ELSIF #baux < 6500.0 THEN
       #Motor := 6500.0;
   ELSE
       #Motor := #baux;
   END_IF;

   #e4 := #e3;
   #e3 := #e2;
   #e2 := #e1;
   #e1 := #e;

   #e4_out_1 := #e4;
   #e3_out_1 := #e3;
   #e2_out_1 := #e2;
   #e1_out_1 := #e;

   #u4 := #u3;
   #u3 := #u2;
   #u2 := #u1;
   #u1 := #baux;
   #u4_out_1 := #u4;
   #u3_out_1 := #u3;
   #u2_out_1 := #u2;
   #u1_out_1 := #u1;
END_FUNCTION_BLOCK

FUNCTION "ALARMAS" : Void   // FC1, LAD
{ S7_Optimized_Access := 'TRUE' }
VERSION : 0.1
BEGIN

REGION Network 1
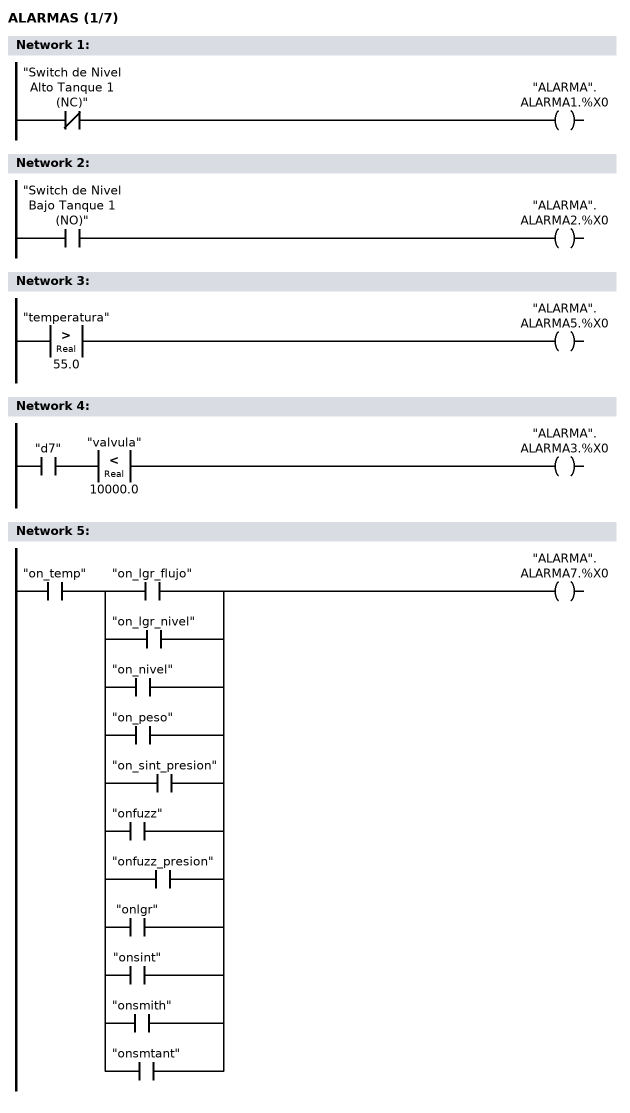
   RUNG wire#powerrail
      I_Contact( "Switch de Nivel Alto Tanque 1 (NC)" )
      Coil( "ALARMA".ALARMA1.%X0 )
   END_RUNG
   // the same network as SCL:
   "ALARMA".ALARMA1.%X0 := NOT "Switch de Nivel Alto Tanque 1 (NC)";
END_REGION

REGION Network 2
   RUNG wire#powerrail
      Contact( "Switch de Nivel Bajo Tanque 1 (NO)" )
      Coil( "ALARMA".ALARMA2.%X0 )
   END_RUNG
   // the same network as SCL:
   "ALARMA".ALARMA2.%X0 := "Switch de Nivel Bajo Tanque 1 (NO)";
END_REGION

REGION Network 3
   RUNG wire#powerrail
      { S7_Templates := "SrcType := Real" } GT_Contact(in1 := "temperatura", in2 := 55.0)
      Coil( "ALARMA".ALARMA5.%X0 )
   END_RUNG
   // the same network as SCL:
   "ALARMA".ALARMA5.%X0 := "temperatura" > 55.0;
END_REGION

REGION Network 4
   RUNG wire#powerrail
      Contact( "d7" )
      { S7_Templates := "SrcType := Real" } LT_Contact(in1 := "valvula", in2 := 10000.0)
      Coil( "ALARMA".ALARMA3.%X0 )
   END_RUNG
   // the same network as SCL:
   "ALARMA".ALARMA3.%X0 := "d7" AND ("valvula" < 10000.0);
END_REGION

REGION Network 5
   RUNG wire#powerrail
      Contact( "on_temp" )
      wire#w1
      Contact( "on_lgr_flujo" )
      wire#w2
      Coil( "ALARMA".ALARMA7.%X0 )
   END_RUNG
   RUNG wire#w1
      Contact( "on_lgr_nivel" )
   END_RUNG wire#w2
   RUNG wire#w1
      Contact( "on_nivel" )
   END_RUNG wire#w2
   RUNG wire#w1
      Contact( "on_peso" )
   END_RUNG wire#w2
   RUNG wire#w1
      Contact( "on_sint_presion" )
   END_RUNG wire#w2
   RUNG wire#w1
      Contact( "onfuzz" )
   END_RUNG wire#w2
   RUNG wire#w1
      Contact( "onfuzz_presion" )
   END_RUNG wire#w2
   RUNG wire#w1
      Contact( "onlgr" )
   END_RUNG wire#w2
   RUNG wire#w1
      Contact( "onsint" )
   END_RUNG wire#w2
   RUNG wire#w1
      Contact( "onsmith" )
   END_RUNG wire#w2
   RUNG wire#w1
      Contact( "onsmtant" )
   END_RUNG wire#w2
   // the same network as SCL:
   "ALARMA".ALARMA7.%X0 := "on_temp" AND ("on_lgr_flujo" OR "on_lgr_nivel" OR "on_nivel" OR "on_peso" OR "on_sint_presion" OR "onfuzz" OR "onfuzz_presion" OR "onlgr" OR "onsint" OR "onsmith" OR "onsmtant");
END_REGION

REGION Network 6
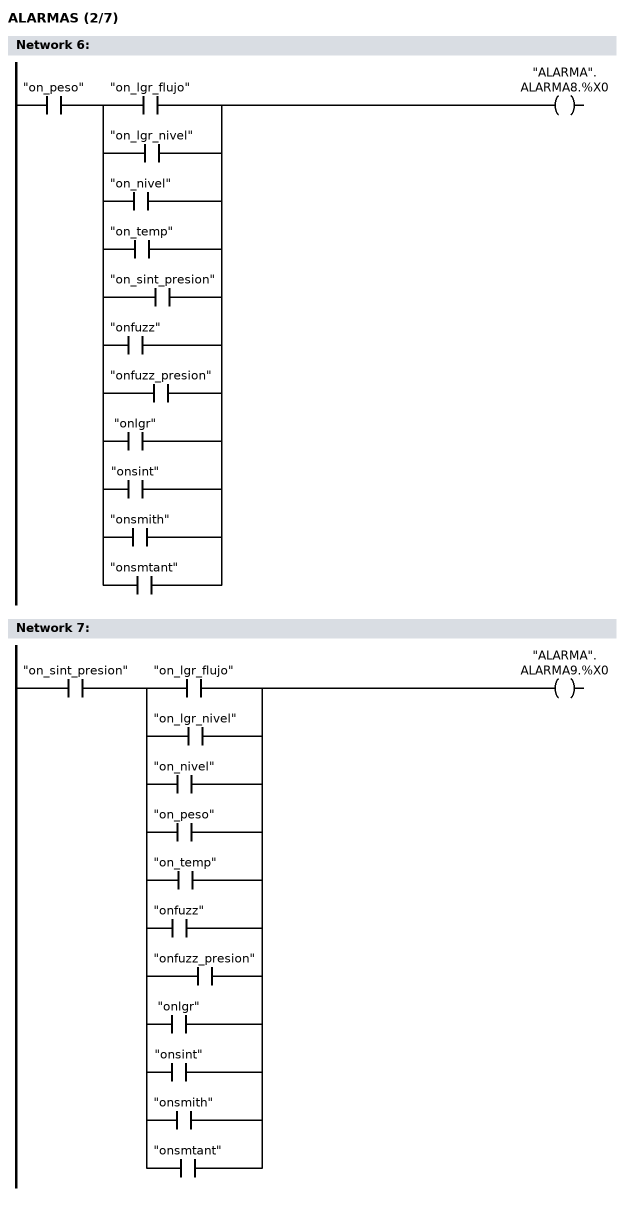
   RUNG wire#powerrail
      Contact( "on_peso" )
      wire#w1
      Contact( "on_lgr_flujo" )
      wire#w2
      Coil( "ALARMA".ALARMA8.%X0 )
   END_RUNG
   RUNG wire#w1
      Contact( "on_lgr_nivel" )
   END_RUNG wire#w2
   RUNG wire#w1
      Contact( "on_nivel" )
   END_RUNG wire#w2
   RUNG wire#w1
      Contact( "on_temp" )
   END_RUNG wire#w2
   RUNG wire#w1
      Contact( "on_sint_presion" )
   END_RUNG wire#w2
   RUNG wire#w1
      Contact( "onfuzz" )
   END_RUNG wire#w2
   RUNG wire#w1
      Contact( "onfuzz_presion" )
   END_RUNG wire#w2
   RUNG wire#w1
      Contact( "onlgr" )
   END_RUNG wire#w2
   RUNG wire#w1
      Contact( "onsint" )
   END_RUNG wire#w2
   RUNG wire#w1
      Contact( "onsmith" )
   END_RUNG wire#w2
   RUNG wire#w1
      Contact( "onsmtant" )
   END_RUNG wire#w2
   // the same network as SCL:
   "ALARMA".ALARMA8.%X0 := "on_peso" AND ("on_lgr_flujo" OR "on_lgr_nivel" OR "on_nivel" OR "on_temp" OR "on_sint_presion" OR "onfuzz" OR "onfuzz_presion" OR "onlgr" OR "onsint" OR "onsmith" OR "onsmtant");
END_REGION

REGION Network 7
   RUNG wire#powerrail
      Contact( "on_sint_presion" )
      wire#w1
      Contact( "on_lgr_flujo" )
      wire#w2
      Coil( "ALARMA".ALARMA9.%X0 )
   END_RUNG
   RUNG wire#w1
      Contact( "on_lgr_nivel" )
   END_RUNG wire#w2
   RUNG wire#w1
      Contact( "on_nivel" )
   END_RUNG wire#w2
   RUNG wire#w1
      Contact( "on_peso" )
   END_RUNG wire#w2
   RUNG wire#w1
      Contact( "on_temp" )
   END_RUNG wire#w2
   RUNG wire#w1
      Contact( "onfuzz" )
   END_RUNG wire#w2
   RUNG wire#w1
      Contact( "onfuzz_presion" )
   END_RUNG wire#w2
   RUNG wire#w1
      Contact( "onlgr" )
   END_RUNG wire#w2
   RUNG wire#w1
      Contact( "onsint" )
   END_RUNG wire#w2
   RUNG wire#w1
      Contact( "onsmith" )
   END_RUNG wire#w2
   RUNG wire#w1
      Contact( "onsmtant" )
   END_RUNG wire#w2
   // the same network as SCL:
   "ALARMA".ALARMA9.%X0 := "on_sint_presion" AND ("on_lgr_flujo" OR "on_lgr_nivel" OR "on_nivel" OR "on_peso" OR "on_temp" OR "onfuzz" OR "onfuzz_presion" OR "onlgr" OR "onsint" OR "onsmith" OR "onsmtant");
END_REGION

REGION Network 8
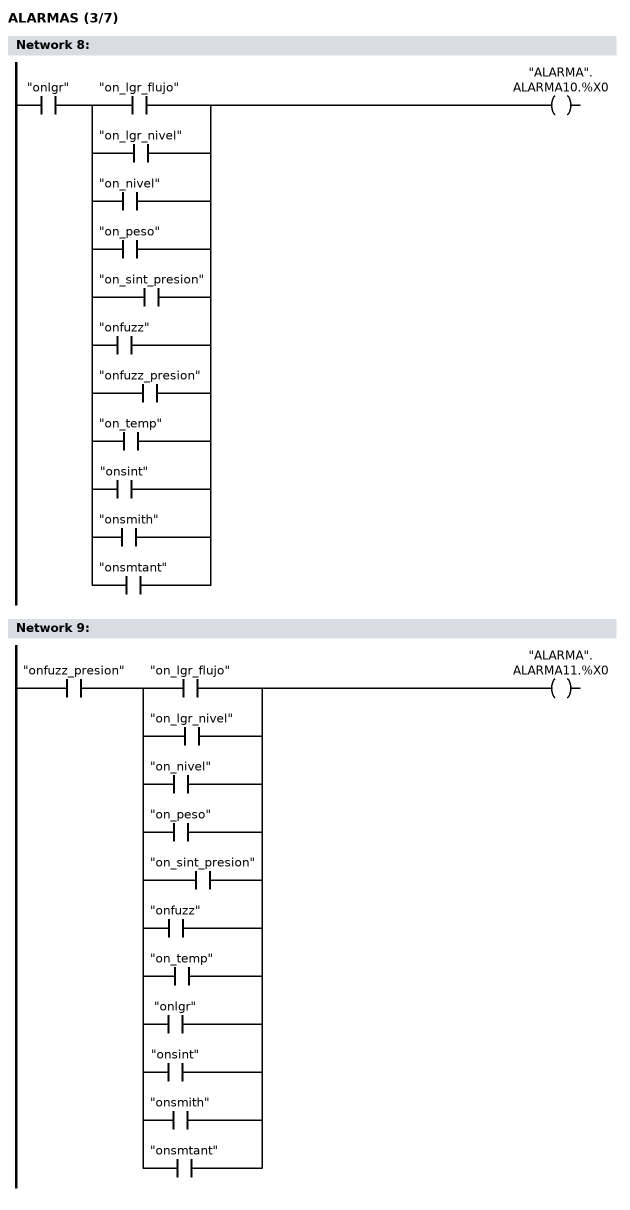
   RUNG wire#powerrail
      Contact( "onlgr" )
      wire#w1
      Contact( "on_lgr_flujo" )
      wire#w2
      Coil( "ALARMA".ALARMA10.%X0 )
   END_RUNG
   RUNG wire#w1
      Contact( "on_lgr_nivel" )
   END_RUNG wire#w2
   RUNG wire#w1
      Contact( "on_nivel" )
   END_RUNG wire#w2
   RUNG wire#w1
      Contact( "on_peso" )
   END_RUNG wire#w2
   RUNG wire#w1
      Contact( "on_sint_presion" )
   END_RUNG wire#w2
   RUNG wire#w1
      Contact( "onfuzz" )
   END_RUNG wire#w2
   RUNG wire#w1
      Contact( "onfuzz_presion" )
   END_RUNG wire#w2
   RUNG wire#w1
      Contact( "on_temp" )
   END_RUNG wire#w2
   RUNG wire#w1
      Contact( "onsint" )
   END_RUNG wire#w2
   RUNG wire#w1
      Contact( "onsmith" )
   END_RUNG wire#w2
   RUNG wire#w1
      Contact( "onsmtant" )
   END_RUNG wire#w2
   // the same network as SCL:
   "ALARMA".ALARMA10.%X0 := "onlgr" AND ("on_lgr_flujo" OR "on_lgr_nivel" OR "on_nivel" OR "on_peso" OR "on_sint_presion" OR "onfuzz" OR "onfuzz_presion" OR "on_temp" OR "onsint" OR "onsmith" OR "onsmtant");
END_REGION

REGION Network 9
   RUNG wire#powerrail
      Contact( "onfuzz_presion" )
      wire#w1
      Contact( "on_lgr_flujo" )
      wire#w2
      Coil( "ALARMA".ALARMA11.%X0 )
   END_RUNG
   RUNG wire#w1
      Contact( "on_lgr_nivel" )
   END_RUNG wire#w2
   RUNG wire#w1
      Contact( "on_nivel" )
   END_RUNG wire#w2
   RUNG wire#w1
      Contact( "on_peso" )
   END_RUNG wire#w2
   RUNG wire#w1
      Contact( "on_sint_presion" )
   END_RUNG wire#w2
   RUNG wire#w1
      Contact( "onfuzz" )
   END_RUNG wire#w2
   RUNG wire#w1
      Contact( "on_temp" )
   END_RUNG wire#w2
   RUNG wire#w1
      Contact( "onlgr" )
   END_RUNG wire#w2
   RUNG wire#w1
      Contact( "onsint" )
   END_RUNG wire#w2
   RUNG wire#w1
      Contact( "onsmith" )
   END_RUNG wire#w2
   RUNG wire#w1
      Contact( "onsmtant" )
   END_RUNG wire#w2
   // the same network as SCL:
   "ALARMA".ALARMA11.%X0 := "onfuzz_presion" AND ("on_lgr_flujo" OR "on_lgr_nivel" OR "on_nivel" OR "on_peso" OR "on_sint_presion" OR "onfuzz" OR "on_temp" OR "onlgr" OR "onsint" OR "onsmith" OR "onsmtant");
END_REGION

REGION Network 10
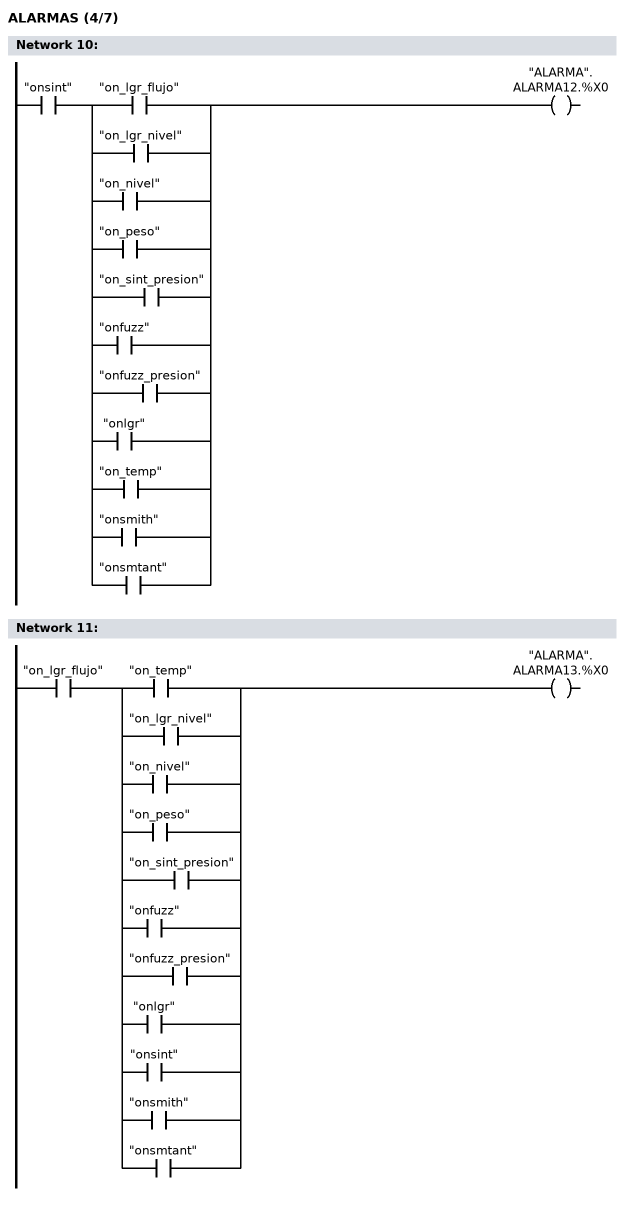
   RUNG wire#powerrail
      Contact( "onsint" )
      wire#w1
      Contact( "on_lgr_flujo" )
      wire#w2
      Coil( "ALARMA".ALARMA12.%X0 )
   END_RUNG
   RUNG wire#w1
      Contact( "on_lgr_nivel" )
   END_RUNG wire#w2
   RUNG wire#w1
      Contact( "on_nivel" )
   END_RUNG wire#w2
   RUNG wire#w1
      Contact( "on_peso" )
   END_RUNG wire#w2
   RUNG wire#w1
      Contact( "on_sint_presion" )
   END_RUNG wire#w2
   RUNG wire#w1
      Contact( "onfuzz" )
   END_RUNG wire#w2
   RUNG wire#w1
      Contact( "onfuzz_presion" )
   END_RUNG wire#w2
   RUNG wire#w1
      Contact( "onlgr" )
   END_RUNG wire#w2
   RUNG wire#w1
      Contact( "on_temp" )
   END_RUNG wire#w2
   RUNG wire#w1
      Contact( "onsmith" )
   END_RUNG wire#w2
   RUNG wire#w1
      Contact( "onsmtant" )
   END_RUNG wire#w2
   // the same network as SCL:
   "ALARMA".ALARMA12.%X0 := "onsint" AND ("on_lgr_flujo" OR "on_lgr_nivel" OR "on_nivel" OR "on_peso" OR "on_sint_presion" OR "onfuzz" OR "onfuzz_presion" OR "onlgr" OR "on_temp" OR "onsmith" OR "onsmtant");
END_REGION

REGION Network 11
   RUNG wire#powerrail
      Contact( "on_lgr_flujo" )
      wire#w1
      Contact( "on_temp" )
      wire#w2
      Coil( "ALARMA".ALARMA13.%X0 )
   END_RUNG
   RUNG wire#w1
      Contact( "on_lgr_nivel" )
   END_RUNG wire#w2
   RUNG wire#w1
      Contact( "on_nivel" )
   END_RUNG wire#w2
   RUNG wire#w1
      Contact( "on_peso" )
   END_RUNG wire#w2
   RUNG wire#w1
      Contact( "on_sint_presion" )
   END_RUNG wire#w2
   RUNG wire#w1
      Contact( "onfuzz" )
   END_RUNG wire#w2
   RUNG wire#w1
      Contact( "onfuzz_presion" )
   END_RUNG wire#w2
   RUNG wire#w1
      Contact( "onlgr" )
   END_RUNG wire#w2
   RUNG wire#w1
      Contact( "onsint" )
   END_RUNG wire#w2
   RUNG wire#w1
      Contact( "onsmith" )
   END_RUNG wire#w2
   RUNG wire#w1
      Contact( "onsmtant" )
   END_RUNG wire#w2
   // the same network as SCL:
   "ALARMA".ALARMA13.%X0 := "on_lgr_flujo" AND ("on_temp" OR "on_lgr_nivel" OR "on_nivel" OR "on_peso" OR "on_sint_presion" OR "onfuzz" OR "onfuzz_presion" OR "onlgr" OR "onsint" OR "onsmith" OR "onsmtant");
END_REGION

REGION Network 12
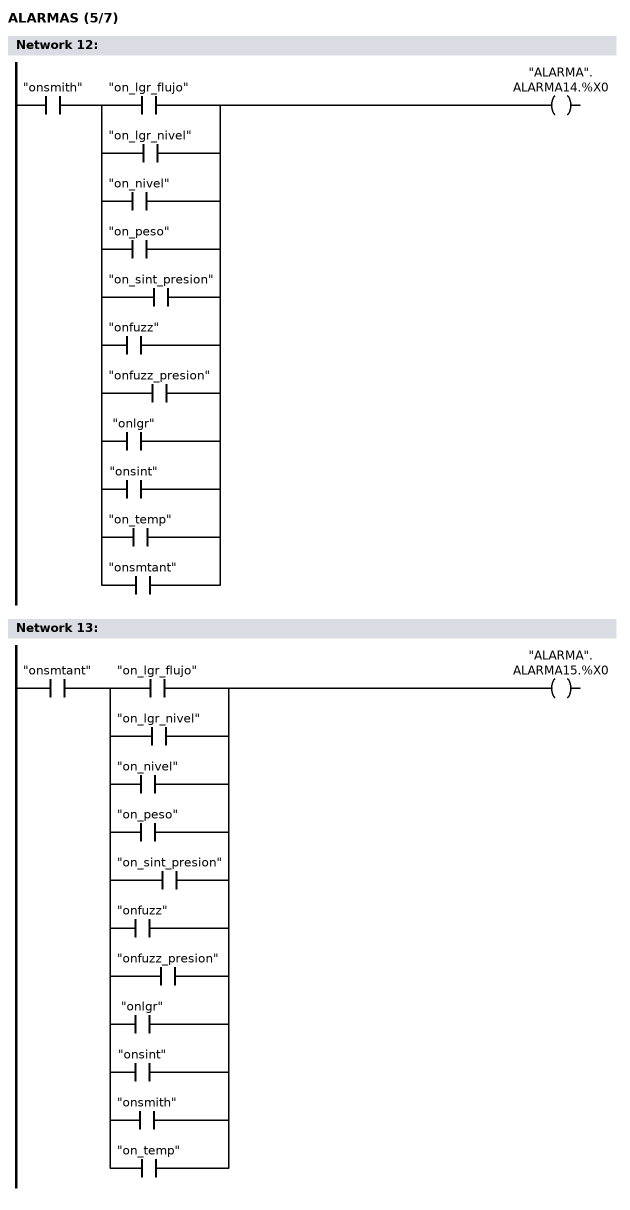
   RUNG wire#powerrail
      Contact( "onsmith" )
      wire#w1
      Contact( "on_lgr_flujo" )
      wire#w2
      Coil( "ALARMA".ALARMA14.%X0 )
   END_RUNG
   RUNG wire#w1
      Contact( "on_lgr_nivel" )
   END_RUNG wire#w2
   RUNG wire#w1
      Contact( "on_nivel" )
   END_RUNG wire#w2
   RUNG wire#w1
      Contact( "on_peso" )
   END_RUNG wire#w2
   RUNG wire#w1
      Contact( "on_sint_presion" )
   END_RUNG wire#w2
   RUNG wire#w1
      Contact( "onfuzz" )
   END_RUNG wire#w2
   RUNG wire#w1
      Contact( "onfuzz_presion" )
   END_RUNG wire#w2
   RUNG wire#w1
      Contact( "onlgr" )
   END_RUNG wire#w2
   RUNG wire#w1
      Contact( "onsint" )
   END_RUNG wire#w2
   RUNG wire#w1
      Contact( "on_temp" )
   END_RUNG wire#w2
   RUNG wire#w1
      Contact( "onsmtant" )
   END_RUNG wire#w2
   // the same network as SCL:
   "ALARMA".ALARMA14.%X0 := "onsmith" AND ("on_lgr_flujo" OR "on_lgr_nivel" OR "on_nivel" OR "on_peso" OR "on_sint_presion" OR "onfuzz" OR "onfuzz_presion" OR "onlgr" OR "onsint" OR "on_temp" OR "onsmtant");
END_REGION

REGION Network 13
   RUNG wire#powerrail
      Contact( "onsmtant" )
      wire#w1
      Contact( "on_lgr_flujo" )
      wire#w2
      Coil( "ALARMA".ALARMA15.%X0 )
   END_RUNG
   RUNG wire#w1
      Contact( "on_lgr_nivel" )
   END_RUNG wire#w2
   RUNG wire#w1
      Contact( "on_nivel" )
   END_RUNG wire#w2
   RUNG wire#w1
      Contact( "on_peso" )
   END_RUNG wire#w2
   RUNG wire#w1
      Contact( "on_sint_presion" )
   END_RUNG wire#w2
   RUNG wire#w1
      Contact( "onfuzz" )
   END_RUNG wire#w2
   RUNG wire#w1
      Contact( "onfuzz_presion" )
   END_RUNG wire#w2
   RUNG wire#w1
      Contact( "onlgr" )
   END_RUNG wire#w2
   RUNG wire#w1
      Contact( "onsint" )
   END_RUNG wire#w2
   RUNG wire#w1
      Contact( "onsmith" )
   END_RUNG wire#w2
   RUNG wire#w1
      Contact( "on_temp" )
   END_RUNG wire#w2
   // the same network as SCL:
   "ALARMA".ALARMA15.%X0 := "onsmtant" AND ("on_lgr_flujo" OR "on_lgr_nivel" OR "on_nivel" OR "on_peso" OR "on_sint_presion" OR "onfuzz" OR "onfuzz_presion" OR "onlgr" OR "onsint" OR "onsmith" OR "on_temp");
END_REGION

REGION Network 14
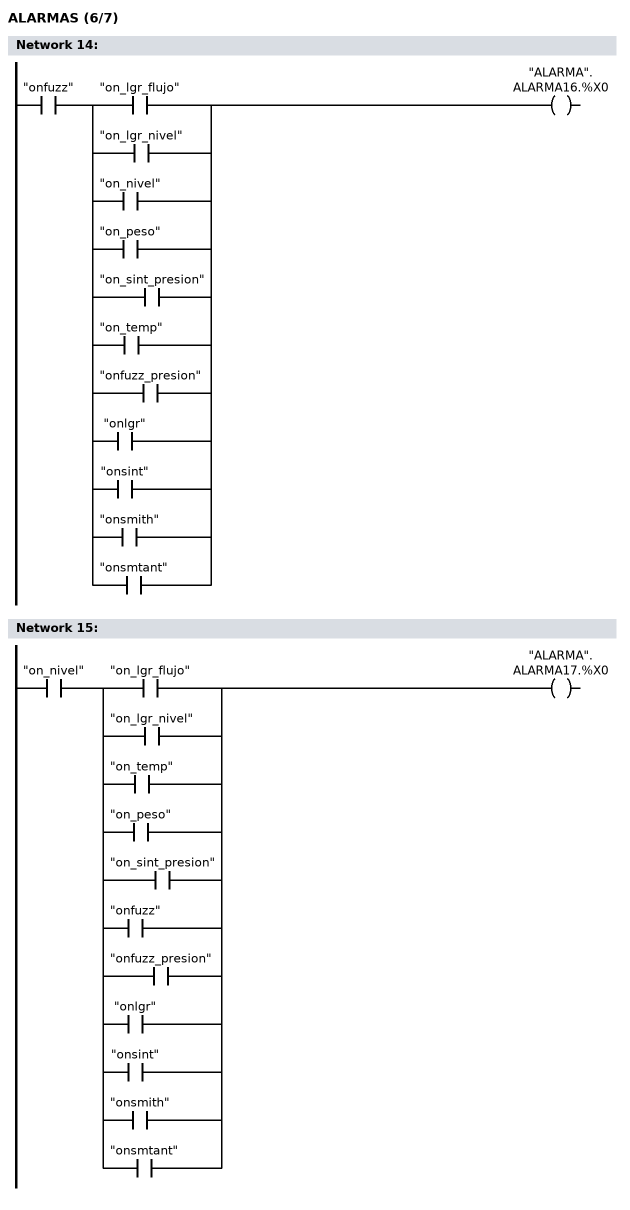
   RUNG wire#powerrail
      Contact( "onfuzz" )
      wire#w1
      Contact( "on_lgr_flujo" )
      wire#w2
      Coil( "ALARMA".ALARMA16.%X0 )
   END_RUNG
   RUNG wire#w1
      Contact( "on_lgr_nivel" )
   END_RUNG wire#w2
   RUNG wire#w1
      Contact( "on_nivel" )
   END_RUNG wire#w2
   RUNG wire#w1
      Contact( "on_peso" )
   END_RUNG wire#w2
   RUNG wire#w1
      Contact( "on_sint_presion" )
   END_RUNG wire#w2
   RUNG wire#w1
      Contact( "on_temp" )
   END_RUNG wire#w2
   RUNG wire#w1
      Contact( "onfuzz_presion" )
   END_RUNG wire#w2
   RUNG wire#w1
      Contact( "onlgr" )
   END_RUNG wire#w2
   RUNG wire#w1
      Contact( "onsint" )
   END_RUNG wire#w2
   RUNG wire#w1
      Contact( "onsmith" )
   END_RUNG wire#w2
   RUNG wire#w1
      Contact( "onsmtant" )
   END_RUNG wire#w2
   // the same network as SCL:
   "ALARMA".ALARMA16.%X0 := "onfuzz" AND ("on_lgr_flujo" OR "on_lgr_nivel" OR "on_nivel" OR "on_peso" OR "on_sint_presion" OR "on_temp" OR "onfuzz_presion" OR "onlgr" OR "onsint" OR "onsmith" OR "onsmtant");
END_REGION

REGION Network 15
   RUNG wire#powerrail
      Contact( "on_nivel" )
      wire#w1
      Contact( "on_lgr_flujo" )
      wire#w2
      Coil( "ALARMA".ALARMA17.%X0 )
   END_RUNG
   RUNG wire#w1
      Contact( "on_lgr_nivel" )
   END_RUNG wire#w2
   RUNG wire#w1
      Contact( "on_temp" )
   END_RUNG wire#w2
   RUNG wire#w1
      Contact( "on_peso" )
   END_RUNG wire#w2
   RUNG wire#w1
      Contact( "on_sint_presion" )
   END_RUNG wire#w2
   RUNG wire#w1
      Contact( "onfuzz" )
   END_RUNG wire#w2
   RUNG wire#w1
      Contact( "onfuzz_presion" )
   END_RUNG wire#w2
   RUNG wire#w1
      Contact( "onlgr" )
   END_RUNG wire#w2
   RUNG wire#w1
      Contact( "onsint" )
   END_RUNG wire#w2
   RUNG wire#w1
      Contact( "onsmith" )
   END_RUNG wire#w2
   RUNG wire#w1
      Contact( "onsmtant" )
   END_RUNG wire#w2
   // the same network as SCL:
   "ALARMA".ALARMA17.%X0 := "on_nivel" AND ("on_lgr_flujo" OR "on_lgr_nivel" OR "on_temp" OR "on_peso" OR "on_sint_presion" OR "onfuzz" OR "onfuzz_presion" OR "onlgr" OR "onsint" OR "onsmith" OR "onsmtant");
END_REGION

REGION Network 16
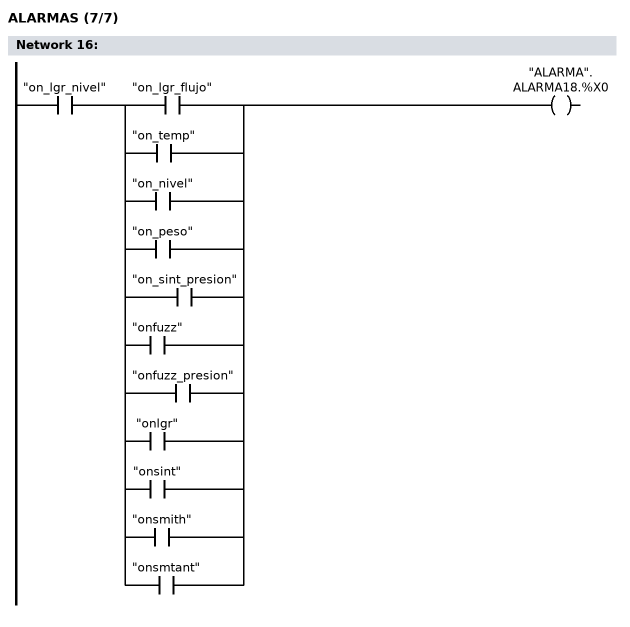
   RUNG wire#powerrail
      Contact( "on_lgr_nivel" )
      wire#w1
      Contact( "on_lgr_flujo" )
      wire#w2
      Coil( "ALARMA".ALARMA18.%X0 )
   END_RUNG
   RUNG wire#w1
      Contact( "on_temp" )
   END_RUNG wire#w2
   RUNG wire#w1
      Contact( "on_nivel" )
   END_RUNG wire#w2
   RUNG wire#w1
      Contact( "on_peso" )
   END_RUNG wire#w2
   RUNG wire#w1
      Contact( "on_sint_presion" )
   END_RUNG wire#w2
   RUNG wire#w1
      Contact( "onfuzz" )
   END_RUNG wire#w2
   RUNG wire#w1
      Contact( "onfuzz_presion" )
   END_RUNG wire#w2
   RUNG wire#w1
      Contact( "onlgr" )
   END_RUNG wire#w2
   RUNG wire#w1
      Contact( "onsint" )
   END_RUNG wire#w2
   RUNG wire#w1
      Contact( "onsmith" )
   END_RUNG wire#w2
   RUNG wire#w1
      Contact( "onsmtant" )
   END_RUNG wire#w2
   // the same network as SCL:
   "ALARMA".ALARMA18.%X0 := "on_lgr_nivel" AND ("on_lgr_flujo" OR "on_temp" OR "on_nivel" OR "on_peso" OR "on_sint_presion" OR "onfuzz" OR "onfuzz_presion" OR "onlgr" OR "onsint" OR "onsmith" OR "onsmtant");
END_REGION
END_FUNCTION

FUNCTION "ENTRADAS_ANALOGAS" : Void   // FC3, LAD
TITLE = ESCALIACIÓN DE ENTRADAS ANALOGAS
{ S7_Optimized_Access := 'TRUE' }
VERSION : 0.1
BEGIN

REGION Network 1: ENTRADAS ANALOGAS - VELOCIDAD VARIADOR
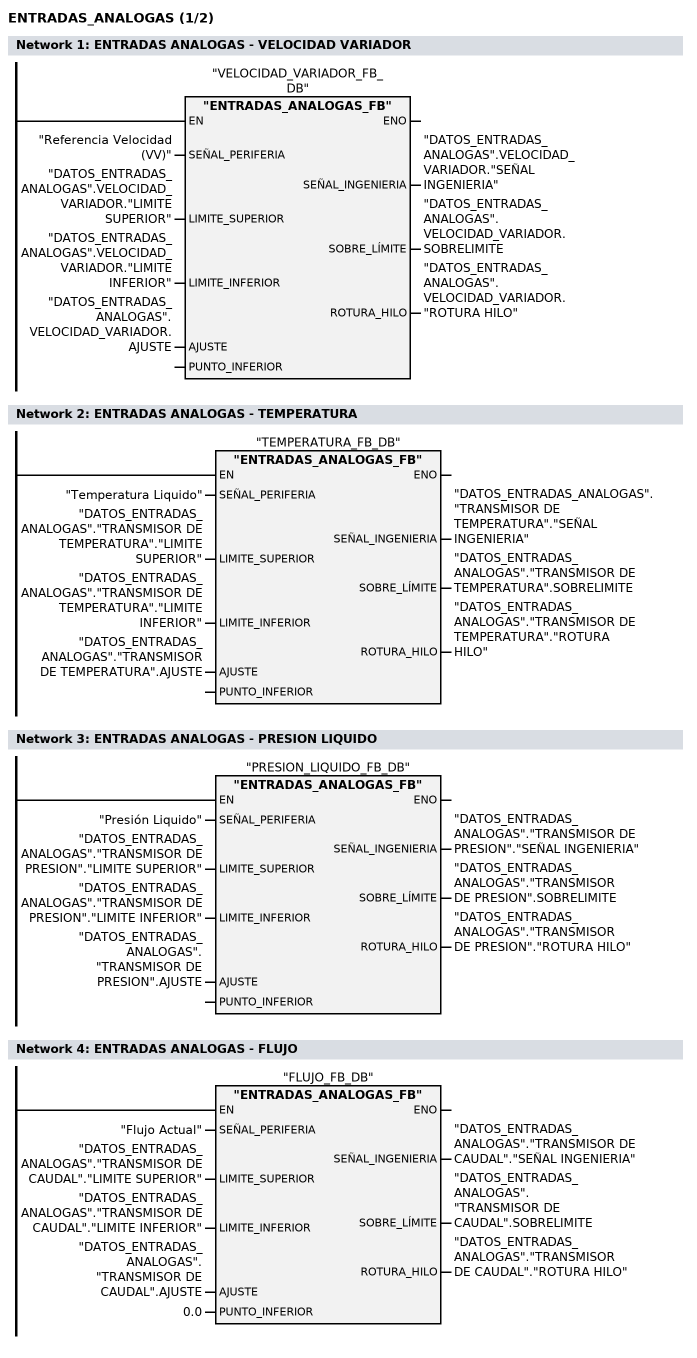
   RUNG wire#powerrail
      "VELOCIDAD_VARIADOR_FB_DB"(SEÑAL_PERIFERIA := "Referencia Velocidad (VV)", LIMITE_SUPERIOR := "DATOS_ENTRADAS_ANALOGAS".VELOCIDAD_VARIADOR."LIMITE SUPERIOR", LIMITE_INFERIOR := "DATOS_ENTRADAS_ANALOGAS".VELOCIDAD_VARIADOR."LIMITE INFERIOR", AJUSTE := "DATOS_ENTRADAS_ANALOGAS".VELOCIDAD_VARIADOR.AJUSTE, PUNTO_INFERIOR :=, SEÑAL_INGENIERIA => "DATOS_ENTRADAS_ANALOGAS".VELOCIDAD_VARIADOR."SEÑAL INGENIERIA", SOBRE_LÍMITE => "DATOS_ENTRADAS_ANALOGAS".VELOCIDAD_VARIADOR.SOBRELIMITE, ROTURA_HILO => "DATOS_ENTRADAS_ANALOGAS".VELOCIDAD_VARIADOR."ROTURA HILO")
   END_RUNG
   // the same network as SCL:
   "VELOCIDAD_VARIADOR_FB_DB"(SEÑAL_PERIFERIA := "Referencia Velocidad (VV)",   // "ENTRADAS_ANALOGAS_FB"
                           LIMITE_SUPERIOR := "DATOS_ENTRADAS_ANALOGAS".VELOCIDAD_VARIADOR."LIMITE SUPERIOR",
                           LIMITE_INFERIOR := "DATOS_ENTRADAS_ANALOGAS".VELOCIDAD_VARIADOR."LIMITE INFERIOR",
                           AJUSTE := "DATOS_ENTRADAS_ANALOGAS".VELOCIDAD_VARIADOR.AJUSTE,
                           SEÑAL_INGENIERIA => "DATOS_ENTRADAS_ANALOGAS".VELOCIDAD_VARIADOR."SEÑAL INGENIERIA",
                           SOBRE_LÍMITE => "DATOS_ENTRADAS_ANALOGAS".VELOCIDAD_VARIADOR.SOBRELIMITE,
                           ROTURA_HILO => "DATOS_ENTRADAS_ANALOGAS".VELOCIDAD_VARIADOR."ROTURA HILO");
END_REGION

REGION Network 2: ENTRADAS ANALOGAS - TEMPERATURA
   RUNG wire#powerrail
      "TEMPERATURA_FB_DB"(SEÑAL_PERIFERIA := "Temperatura Liquido", LIMITE_SUPERIOR := "DATOS_ENTRADAS_ANALOGAS"."TRANSMISOR DE TEMPERATURA"."LIMITE SUPERIOR", LIMITE_INFERIOR := "DATOS_ENTRADAS_ANALOGAS"."TRANSMISOR DE TEMPERATURA"."LIMITE INFERIOR", AJUSTE := "DATOS_ENTRADAS_ANALOGAS"."TRANSMISOR DE TEMPERATURA".AJUSTE, PUNTO_INFERIOR :=, SEÑAL_INGENIERIA => "DATOS_ENTRADAS_ANALOGAS"."TRANSMISOR DE TEMPERATURA"."SEÑAL INGENIERIA", SOBRE_LÍMITE => "DATOS_ENTRADAS_ANALOGAS"."TRANSMISOR DE TEMPERATURA".SOBRELIMITE, ROTURA_HILO => "DATOS_ENTRADAS_ANALOGAS"."TRANSMISOR DE TEMPERATURA"."ROTURA HILO")
   END_RUNG
   // the same network as SCL:
   "TEMPERATURA_FB_DB"(SEÑAL_PERIFERIA := "Temperatura Liquido",   // "ENTRADAS_ANALOGAS_FB"
                       LIMITE_SUPERIOR := "DATOS_ENTRADAS_ANALOGAS"."TRANSMISOR DE TEMPERATURA"."LIMITE SUPERIOR",
                       LIMITE_INFERIOR := "DATOS_ENTRADAS_ANALOGAS"."TRANSMISOR DE TEMPERATURA"."LIMITE INFERIOR",
                       AJUSTE := "DATOS_ENTRADAS_ANALOGAS"."TRANSMISOR DE TEMPERATURA".AJUSTE,
                       SEÑAL_INGENIERIA => "DATOS_ENTRADAS_ANALOGAS"."TRANSMISOR DE TEMPERATURA"."SEÑAL INGENIERIA",
                       SOBRE_LÍMITE => "DATOS_ENTRADAS_ANALOGAS"."TRANSMISOR DE TEMPERATURA".SOBRELIMITE,
                       ROTURA_HILO => "DATOS_ENTRADAS_ANALOGAS"."TRANSMISOR DE TEMPERATURA"."ROTURA HILO");
END_REGION

REGION Network 3: ENTRADAS ANALOGAS - PRESION LIQUIDO
   RUNG wire#powerrail
      "PRESION_LIQUIDO_FB_DB"(SEÑAL_PERIFERIA := "Presión Liquido", LIMITE_SUPERIOR := "DATOS_ENTRADAS_ANALOGAS"."TRANSMISOR DE PRESION"."LIMITE SUPERIOR", LIMITE_INFERIOR := "DATOS_ENTRADAS_ANALOGAS"."TRANSMISOR DE PRESION"."LIMITE INFERIOR", AJUSTE := "DATOS_ENTRADAS_ANALOGAS"."TRANSMISOR DE PRESION".AJUSTE, PUNTO_INFERIOR :=, SEÑAL_INGENIERIA => "DATOS_ENTRADAS_ANALOGAS"."TRANSMISOR DE PRESION"."SEÑAL INGENIERIA", SOBRE_LÍMITE => "DATOS_ENTRADAS_ANALOGAS"."TRANSMISOR DE PRESION".SOBRELIMITE, ROTURA_HILO => "DATOS_ENTRADAS_ANALOGAS"."TRANSMISOR DE PRESION"."ROTURA HILO")
   END_RUNG
   // the same network as SCL:
   "PRESION_LIQUIDO_FB_DB"(SEÑAL_PERIFERIA := "Presión Liquido",   // "ENTRADAS_ANALOGAS_FB"
                           LIMITE_SUPERIOR := "DATOS_ENTRADAS_ANALOGAS"."TRANSMISOR DE PRESION"."LIMITE SUPERIOR",
                           LIMITE_INFERIOR := "DATOS_ENTRADAS_ANALOGAS"."TRANSMISOR DE PRESION"."LIMITE INFERIOR",
                           AJUSTE := "DATOS_ENTRADAS_ANALOGAS"."TRANSMISOR DE PRESION".AJUSTE,
                           SEÑAL_INGENIERIA => "DATOS_ENTRADAS_ANALOGAS"."TRANSMISOR DE PRESION"."SEÑAL INGENIERIA",
                           SOBRE_LÍMITE => "DATOS_ENTRADAS_ANALOGAS"."TRANSMISOR DE PRESION".SOBRELIMITE,
                           ROTURA_HILO => "DATOS_ENTRADAS_ANALOGAS"."TRANSMISOR DE PRESION"."ROTURA HILO");
END_REGION

REGION Network 4: ENTRADAS ANALOGAS - FLUJO
   RUNG wire#powerrail
      "FLUJO_FB_DB"(SEÑAL_PERIFERIA := "Flujo Actual", LIMITE_SUPERIOR := "DATOS_ENTRADAS_ANALOGAS"."TRANSMISOR DE CAUDAL"."LIMITE SUPERIOR", LIMITE_INFERIOR := "DATOS_ENTRADAS_ANALOGAS"."TRANSMISOR DE CAUDAL"."LIMITE INFERIOR", AJUSTE := "DATOS_ENTRADAS_ANALOGAS"."TRANSMISOR DE CAUDAL".AJUSTE, PUNTO_INFERIOR := 0.0, SEÑAL_INGENIERIA => "DATOS_ENTRADAS_ANALOGAS"."TRANSMISOR DE CAUDAL"."SEÑAL INGENIERIA", SOBRE_LÍMITE => "DATOS_ENTRADAS_ANALOGAS"."TRANSMISOR DE CAUDAL".SOBRELIMITE, ROTURA_HILO => "DATOS_ENTRADAS_ANALOGAS"."TRANSMISOR DE CAUDAL"."ROTURA HILO")
   END_RUNG
   // the same network as SCL:
   "FLUJO_FB_DB"(SEÑAL_PERIFERIA := "Flujo Actual",   // "ENTRADAS_ANALOGAS_FB"
                 LIMITE_SUPERIOR := "DATOS_ENTRADAS_ANALOGAS"."TRANSMISOR DE CAUDAL"."LIMITE SUPERIOR",
                 LIMITE_INFERIOR := "DATOS_ENTRADAS_ANALOGAS"."TRANSMISOR DE CAUDAL"."LIMITE INFERIOR",
                 AJUSTE := "DATOS_ENTRADAS_ANALOGAS"."TRANSMISOR DE CAUDAL".AJUSTE,
                 PUNTO_INFERIOR := 0.0,
                 SEÑAL_INGENIERIA => "DATOS_ENTRADAS_ANALOGAS"."TRANSMISOR DE CAUDAL"."SEÑAL INGENIERIA",
                 SOBRE_LÍMITE => "DATOS_ENTRADAS_ANALOGAS"."TRANSMISOR DE CAUDAL".SOBRELIMITE,
                 ROTURA_HILO => "DATOS_ENTRADAS_ANALOGAS"."TRANSMISOR DE CAUDAL"."ROTURA HILO");
END_REGION

REGION Network 5: ENTRADAS ANALOGAS - NIVEL
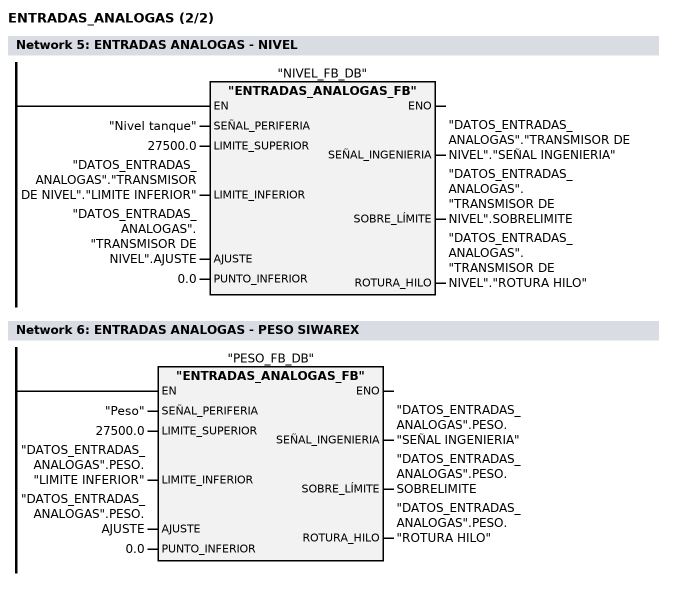
   RUNG wire#powerrail
      "NIVEL_FB_DB"(SEÑAL_PERIFERIA := "Nivel tanque", LIMITE_SUPERIOR := 27500.0, LIMITE_INFERIOR := "DATOS_ENTRADAS_ANALOGAS"."TRANSMISOR DE NIVEL"."LIMITE INFERIOR", AJUSTE := "DATOS_ENTRADAS_ANALOGAS"."TRANSMISOR DE NIVEL".AJUSTE, PUNTO_INFERIOR := 0.0, SEÑAL_INGENIERIA => "DATOS_ENTRADAS_ANALOGAS"."TRANSMISOR DE NIVEL"."SEÑAL INGENIERIA", SOBRE_LÍMITE => "DATOS_ENTRADAS_ANALOGAS"."TRANSMISOR DE NIVEL".SOBRELIMITE, ROTURA_HILO => "DATOS_ENTRADAS_ANALOGAS"."TRANSMISOR DE NIVEL"."ROTURA HILO")
   END_RUNG
   // the same network as SCL:
   "NIVEL_FB_DB"(SEÑAL_PERIFERIA := "Nivel tanque",   // "ENTRADAS_ANALOGAS_FB"
                 LIMITE_SUPERIOR := 27500.0,
                 LIMITE_INFERIOR := "DATOS_ENTRADAS_ANALOGAS"."TRANSMISOR DE NIVEL"."LIMITE INFERIOR",
                 AJUSTE := "DATOS_ENTRADAS_ANALOGAS"."TRANSMISOR DE NIVEL".AJUSTE,
                 PUNTO_INFERIOR := 0.0,
                 SEÑAL_INGENIERIA => "DATOS_ENTRADAS_ANALOGAS"."TRANSMISOR DE NIVEL"."SEÑAL INGENIERIA",
                 SOBRE_LÍMITE => "DATOS_ENTRADAS_ANALOGAS"."TRANSMISOR DE NIVEL".SOBRELIMITE,
                 ROTURA_HILO => "DATOS_ENTRADAS_ANALOGAS"."TRANSMISOR DE NIVEL"."ROTURA HILO");
END_REGION

REGION Network 6: ENTRADAS ANALOGAS - PESO SIWAREX
   RUNG wire#powerrail
      "PESO_FB_DB"(SEÑAL_PERIFERIA := "Peso", LIMITE_SUPERIOR := 27500.0, LIMITE_INFERIOR := "DATOS_ENTRADAS_ANALOGAS".PESO."LIMITE INFERIOR", AJUSTE := "DATOS_ENTRADAS_ANALOGAS".PESO.AJUSTE, PUNTO_INFERIOR := 0.0, SEÑAL_INGENIERIA => "DATOS_ENTRADAS_ANALOGAS".PESO."SEÑAL INGENIERIA", SOBRE_LÍMITE => "DATOS_ENTRADAS_ANALOGAS".PESO.SOBRELIMITE, ROTURA_HILO => "DATOS_ENTRADAS_ANALOGAS".PESO."ROTURA HILO")
   END_RUNG
   // the same network as SCL:
   "PESO_FB_DB"(SEÑAL_PERIFERIA := "Peso",   // "ENTRADAS_ANALOGAS_FB"
                LIMITE_SUPERIOR := 27500.0,
                LIMITE_INFERIOR := "DATOS_ENTRADAS_ANALOGAS".PESO."LIMITE INFERIOR",
                AJUSTE := "DATOS_ENTRADAS_ANALOGAS".PESO.AJUSTE,
                PUNTO_INFERIOR := 0.0,
                SEÑAL_INGENIERIA => "DATOS_ENTRADAS_ANALOGAS".PESO."SEÑAL INGENIERIA",
                SOBRE_LÍMITE => "DATOS_ENTRADAS_ANALOGAS".PESO.SOBRELIMITE,
                ROTURA_HILO => "DATOS_ENTRADAS_ANALOGAS".PESO."ROTURA HILO");
END_REGION
END_FUNCTION

FUNCTION "SALIDAS_ANALOGAS" : Void   // FC4, LAD
{ S7_Optimized_Access := 'TRUE' }
VERSION : 0.1
BEGIN

REGION Network 1: SALIDAS ANALOGAS - VELOCIDAD VARIADOR
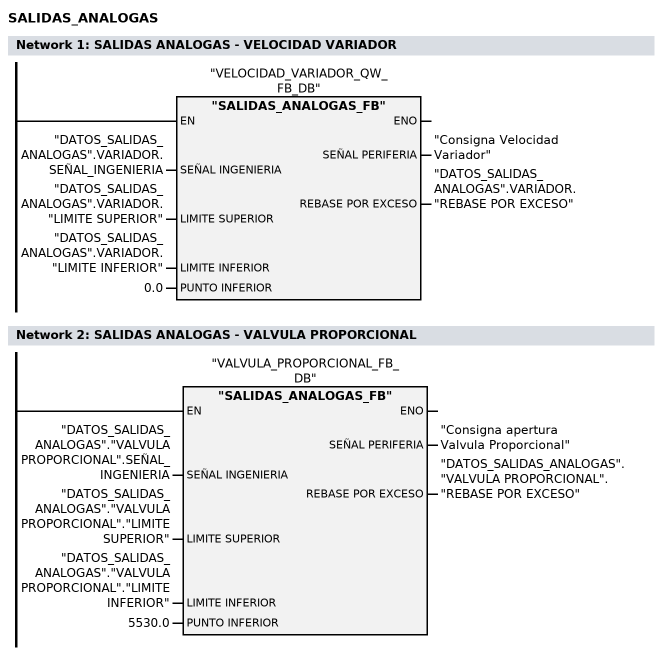
   RUNG wire#powerrail
      "VELOCIDAD_VARIADOR_QW_FB_DB"("SEÑAL INGENIERIA" := "DATOS_SALIDAS_ANALOGAS".VARIADOR.SEÑAL_INGENIERIA, "LIMITE SUPERIOR" := "DATOS_SALIDAS_ANALOGAS".VARIADOR."LIMITE SUPERIOR", "LIMITE INFERIOR" := "DATOS_SALIDAS_ANALOGAS".VARIADOR."LIMITE INFERIOR", "PUNTO INFERIOR" := 0.0, "SEÑAL PERIFERIA" => "Consigna Velocidad Variador", "REBASE POR EXCESO" => "DATOS_SALIDAS_ANALOGAS".VARIADOR."REBASE POR EXCESO")
   END_RUNG
   // the same network as SCL:
   "VELOCIDAD_VARIADOR_QW_FB_DB"("SEÑAL INGENIERIA" := "DATOS_SALIDAS_ANALOGAS".VARIADOR.SEÑAL_INGENIERIA,   // "SALIDAS_ANALOGAS_FB"
                           "LIMITE SUPERIOR" := "DATOS_SALIDAS_ANALOGAS".VARIADOR."LIMITE SUPERIOR",
                           "LIMITE INFERIOR" := "DATOS_SALIDAS_ANALOGAS".VARIADOR."LIMITE INFERIOR",
                           "PUNTO INFERIOR" := 0.0,
                           "SEÑAL PERIFERIA" => "Consigna Velocidad Variador",
                           "REBASE POR EXCESO" => "DATOS_SALIDAS_ANALOGAS".VARIADOR."REBASE POR EXCESO");
END_REGION

REGION Network 2: SALIDAS ANALOGAS - VALVULA PROPORCIONAL
   RUNG wire#powerrail
      "VALVULA_PROPORCIONAL_FB_DB"("SEÑAL INGENIERIA" := "DATOS_SALIDAS_ANALOGAS"."VALVULA PROPORCIONAL".SEÑAL_INGENIERIA, "LIMITE SUPERIOR" := "DATOS_SALIDAS_ANALOGAS"."VALVULA PROPORCIONAL"."LIMITE SUPERIOR", "LIMITE INFERIOR" := "DATOS_SALIDAS_ANALOGAS"."VALVULA PROPORCIONAL"."LIMITE INFERIOR", "PUNTO INFERIOR" := 5530.0, "SEÑAL PERIFERIA" => "Consigna apertura Valvula Proporcional", "REBASE POR EXCESO" => "DATOS_SALIDAS_ANALOGAS"."VALVULA PROPORCIONAL"."REBASE POR EXCESO")
   END_RUNG
   // the same network as SCL:
   "VALVULA_PROPORCIONAL_FB_DB"("SEÑAL INGENIERIA" := "DATOS_SALIDAS_ANALOGAS"."VALVULA PROPORCIONAL".SEÑAL_INGENIERIA,   // "SALIDAS_ANALOGAS_FB"
                           "LIMITE SUPERIOR" := "DATOS_SALIDAS_ANALOGAS"."VALVULA PROPORCIONAL"."LIMITE SUPERIOR",
                           "LIMITE INFERIOR" := "DATOS_SALIDAS_ANALOGAS"."VALVULA PROPORCIONAL"."LIMITE INFERIOR",
                           "PUNTO INFERIOR" := 5530.0,
                           "SEÑAL PERIFERIA" => "Consigna apertura Valvula Proporcional",
                           "REBASE POR EXCESO" => "DATOS_SALIDAS_ANALOGAS"."VALVULA PROPORCIONAL"."REBASE POR EXCESO");
END_REGION
END_FUNCTION

FUNCTION "fuzzyfica" : Void   // FC7, SCL
{ S7_Optimized_Access := 'TRUE' }
VERSION : 0.1
   VAR_INPUT
      crisp : Real;
      vector1 : Real;
      vector2 : Real;
      vector3 : Real;
      vector4 : Real;
   END_VAR
   VAR_OUTPUT
      A_1 : Real;
   END_VAR
   VAR_TEMP
      "a" : Real;
      "B" : Real;
   END_VAR
BEGIN

   IF (#vector1 < #crisp & #crisp < #vector2) THEN
       #B := -1 * (((1 - 0) / (#vector2 - #vector1)) * #vector1);
       #a := (((1 - 0) / (#vector2 - #vector1)) * #crisp) + #B;
       #A_1 := #a;
       RETURN;
   ELSIF (#vector2 < #crisp & #crisp < #vector3) THEN
       #a := 1;
       #A_1 := #a;
       RETURN;
   ELSIF (#vector3 < #crisp & #crisp < #vector4) THEN
       #B := (((1 - 0) / (#vector2 - #vector1)) * #vector4);
       #a := (((0 - 1) / (#vector4 - #vector3)) * #crisp) + #B;
       #A_1 := #a;
       RETURN;
   ELSE
       #a := 0;
       #A_1 := #a;
       RETURN;
   END_IF;
END_FUNCTION

ORGANIZATION_BLOCK "Main"   // OB1, LAD, ProgramCycle
TITLE = "Main Program Sweep (Cycle)"
{ S7_Optimized_Access := 'TRUE' }
VERSION : 0.1
   VAR_INPUT
      Initial_Call : Bool;   // Initial call of this OB
      Remanence : Bool;   // =True, if remanent data are available
   END_VAR
   VAR_TEMP
      NIVELTV : Int;
      "a" : Real;
      MARCA : Bool;
   END_VAR
   VAR_TEMP   // added for the SCL form of the ladder/FBD networks
      _w1 : Bool;
   END_VAR
BEGIN

REGION Network 1: LINEALIZACION SENSORES
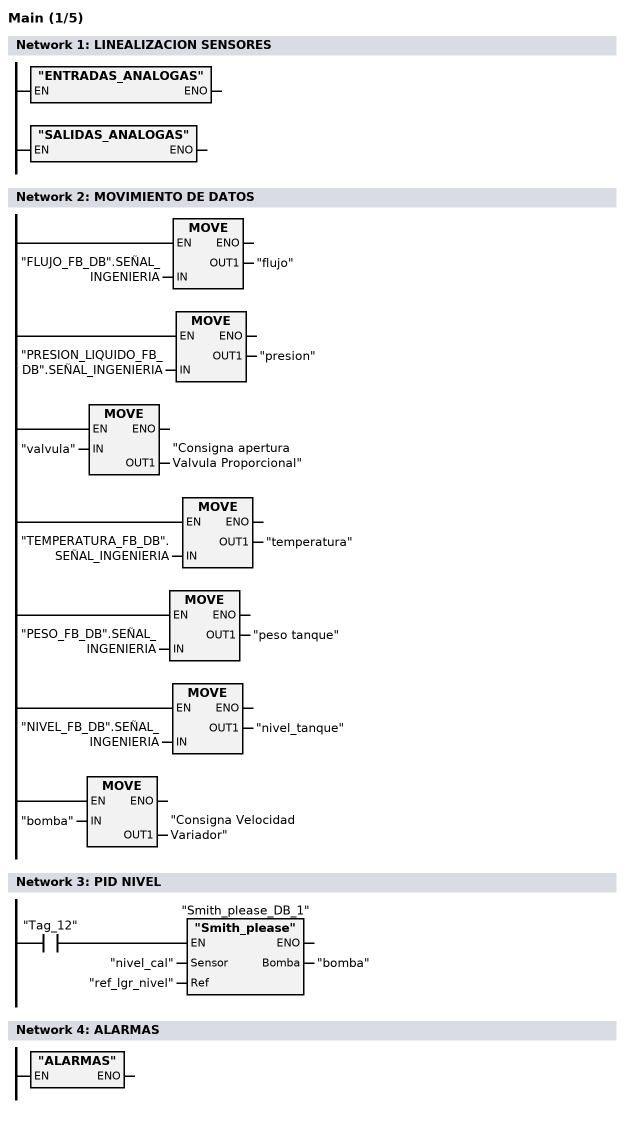
   RUNG wire#powerrail
      "ENTRADAS_ANALOGAS"()
   END_RUNG
   RUNG wire#powerrail
      "SALIDAS_ANALOGAS"()
   END_RUNG
   // the same network as SCL:
   "ENTRADAS_ANALOGAS"();
   "SALIDAS_ANALOGAS"();
END_REGION

